SPLINE
SPL {X  -159.452, Y  +378.767, Z    +0.000, E1   +11.887, E3 +78162.676}
SPL {X  -159.840, Y  +384.856, Z    +0.000, E1    +7.126, E3 +78181.648}
SPL {X  -159.991, Y  +390.336, Z    +0.000, E1    +2.803, E3 +78195.471}
SPL {X  -160.000, Y  +403.532, Z    +0.000, E1    -6.523, E3 +78213.191}
SPL {X  -160.000, Y  +409.023, Z    +0.000, E1   -10.003, E3 +78223.965}
SPL {X  -160.000, Y  +418.032, Z    +0.000, E1   -14.569, E3 +78248.824}
SPL {X  -160.000, Y  +420.561, Z    +0.000, E1   -14.816, E3 +78266.304}
SPL {X  -160.000, Y  +422.801, Z    +0.000, E1   -14.823, E3 +78284.253}
SPL {X  -160.000, Y  +425.518, Z    +0.000, E1   -14.845, E3 +78306.027}
SPL {X  -160.000, Y  +428.688, Z    +0.000, E1   -14.854, E3 +78331.435}
SPL {X  -160.000, Y  +431.971, Z    +0.000, E1   -14.849, E3 +78357.904}
SPL {X  -160.000, Y  +435.345, Z    +0.000, E1   -14.857, E3 +78384.954}
SPL {X  -160.000, Y  +438.732, Z    +0.000, E1   -14.858, E3 +78412.103}
SPL {X  -160.000, Y  +441.925, Z    +0.000, E1   -14.848, E3 +78437.773}
SPL {X  -160.000, Y  +444.299, Z    +0.000, E1   -14.809, E3 +78456.958}
SPL {X  -160.000, Y  +446.229, Z    +0.000, E1   -14.820, E3 +78472.377}
SPL {X  -160.000, Y  +448.987, Z    +0.000, E1   -14.868, E3 +78494.313}
SPL {X  -160.000, Y  +452.351, Z    +0.000, E1   -14.871, E3 +78521.289}
SPL {X  -160.000, Y  +455.709, Z    +0.000, E1   -14.880, E3 +78548.103}
SPL {X  -160.000, Y  +458.189, Z    +0.000, E1   -14.832, E3 +78568.105}
SPL {X  -160.000, Y  +459.885, Z    +0.000, E1   -14.825, E3 +78581.776}
SPL {X  -160.000, Y  +462.438, Z    +0.000, E1   -14.868, E3 +78602.186}
SPL {X  -160.000, Y  +465.575, Z    +0.000, E1   -14.849, E3 +78627.494}
SPL {X  -160.000, Y  +468.581, Z    +0.000, E1   -14.841, E3 +78651.726}
SPL {X  -160.000, Y  +471.795, Z    +0.000, E1   -14.854, E3 +78677.514}
SPL {X  -160.000, Y  +475.138, Z    +0.000, E1   -14.853, E3 +78704.364}
SPL {X  -160.000, Y  +477.981, Z    +0.000, E1   -14.823, E3 +78727.284}
SPL {X  -160.000, Y  +480.658, Z    +0.000, E1   -14.835, E3 +78748.760}
SPL {X  -160.000, Y  +483.534, Z    +0.000, E1   -14.838, E3 +78771.855}
SPL {X  -160.000, Y  +486.226, Z    +0.000, E1   -14.823, E3 +78793.520}
SPL {X  -160.000, Y  +488.751, Z    +0.000, E1   -14.827, E3 +78813.793}
SPL {X  -160.000, Y  +491.612, Z    +0.000, E1   -14.844, E3 +78836.716}
SPL {X  -160.000, Y  +494.417, Z    +0.000, E1   -14.827, E3 +78859.306}
SPL {X  -160.000, Y  +496.961, Z    +0.000, E1   -14.824, E3 +78879.750}
SPL {X  -160.000, Y  +499.610, Z    +0.000, E1   -14.830, E3 +78901.023}
SPL {X  -160.000, Y  +502.268, Z    +0.000, E1   -14.832, E3 +78922.292}
SPL {X  -160.000, Y  +505.041, Z    +0.000, E1   -14.849, E3 +78944.455}
SPL {X  -160.000, Y  +507.743, Z    +0.000, E1   -14.842, E3 +78966.078}
SPL {X  -160.000, Y  +510.437, Z    +0.000, E1   -14.860, E3 +78987.592}
SPL {X  -160.000, Y  +513.179, Z    +0.000, E1   -14.849, E3 +79009.640}
SPL {X  -160.000, Y  +515.613, Z    +0.000, E1   -14.829, E3 +79029.310}
SPL {X  -160.000, Y  +518.188, Z    +0.000, E1   -14.845, E3 +79049.939}
SPL {X  -160.000, Y  +520.790, Z    +0.000, E1   -14.839, E3 +79070.768}
SPL {X  -160.000, Y  +523.469, Z    +0.000, E1   -14.855, E3 +79092.216}
SPL {X  -160.000, Y  +526.403, Z    +0.000, E1   -14.858, E3 +79115.753}
SPL {X  -160.000, Y  +529.266, Z    +0.000, E1   -14.848, E3 +79138.760}
SPL {X  -160.000, Y  +531.688, Z    +0.000, E1   -14.826, E3 +79158.310}
SPL {X  -160.000, Y  +534.214, Z    +0.000, E1   -14.841, E3 +79178.573}
SPL {X  -160.000, Y  +537.002, Z    +0.000, E1   -14.839, E3 +79200.991}
SPL {X  -160.000, Y  +539.729, Z    +0.000, E1   -14.840, E3 +79222.803}
SPL {X  -160.000, Y  +542.408, Z    +0.000, E1   -14.839, E3 +79244.356}
SPL {X  -160.000, Y  +545.014, Z    +0.000, E1   -14.831, E3 +79265.301}
SPL {X  -160.000, Y  +547.659, Z    +0.000, E1   -14.839, E3 +79286.515}
SPL {X  -160.000, Y  +550.215, Z    +0.000, E1   -14.827, E3 +79307.080}
SPL {X  -160.000, Y  +552.762, Z    +0.000, E1   -14.836, E3 +79327.499}
SPL {X  -160.000, Y  +555.331, Z    +0.000, E1   -14.837, E3 +79348.040}
SPL {X  -160.000, Y  +558.235, Z    +0.000, E1   -14.869, E3 +79371.203}
SPL {X  -160.000, Y  +561.088, Z    +0.000, E1   -14.848, E3 +79394.122}
SPL {X  -160.000, Y  +563.693, Z    +0.000, E1   -14.852, E3 +79414.982}
SPL {X  -160.000, Y  +566.560, Z    +0.000, E1   -14.865, E3 +79437.960}
SPL {X  -160.000, Y  +569.305, Z    +0.000, E1   -14.848, E3 +79459.988}
SPL {X  -160.000, Y  +571.769, Z    +0.000, E1   -14.852, E3 +79479.734}
SPL {X  -160.000, Y  +574.366, Z    +0.000, E1   -14.855, E3 +79500.521}
SPL {X  -160.000, Y  +577.037, Z    +0.000, E1   -14.859, E3 +79521.921}
SPL {X  -160.000, Y  +579.855, Z    +0.000, E1   -14.869, E3 +79544.448}
SPL {X  -160.000, Y  +582.456, Z    +0.000, E1   -14.854, E3 +79565.308}
SPL {X  -160.000, Y  +585.083, Z    +0.000, E1   -14.866, E3 +79586.358}
SPL {X  -160.000, Y  +587.675, Z    +0.000, E1   -14.853, E3 +79607.148}
SPL {X  -160.000, Y  +590.216, Z    +0.000, E1   -14.864, E3 +79627.468}
SPL {X  -160.000, Y  +592.848, Z    +0.000, E1   -14.865, E3 +79648.519}
SPL {X  -160.000, Y  +595.342, Z    +0.000, E1   -14.848, E3 +79668.696}
SPL {X  -160.000, Y  +597.995, Z    +0.000, E1   -14.848, E3 +79690.036}
SPL {X  -160.000, Y  +600.731, Z    +0.000, E1   -14.846, E3 +79711.988}
SPL {X  -160.000, Y  +603.404, Z    +0.000, E1   -14.846, E3 +79733.424}
SPL {X  -160.000, Y  +605.923, Z    +0.000, E1   -14.838, E3 +79753.664}
SPL {X  -160.000, Y  +608.492, Z    +0.000, E1   -14.846, E3 +79774.268}
SPL {X  -160.000, Y  +611.345, Z    +0.000, E1   -14.856, E3 +79797.126}
SPL {X  -160.000, Y  +614.087, Z    +0.000, E1   -14.839, E3 +79819.186}
SPL {X  -160.000, Y  +616.566, Z    +0.000, E1   -14.839, E3 +79839.079}
SPL {X  -160.000, Y  +619.350, Z    +0.000, E1   -14.855, E3 +79861.367}
SPL {X  -160.000, Y  +622.198, Z    +0.000, E1   -14.846, E3 +79884.252}
SPL {X  -160.000, Y  +624.642, Z    +0.000, E1   -14.829, E3 +79903.925}
SPL {X  -160.000, Y  +627.119, Z    +0.000, E1   -14.843, E3 +79923.764}
SPL {X  -160.000, Y  +629.682, Z    +0.000, E1   -14.838, E3 +79944.333}
SPL {X  -160.000, Y  +632.223, Z    +0.000, E1   -14.841, E3 +79964.725}
SPL {X  -160.000, Y  +634.941, Z    +0.000, E1   -14.846, E3 +79986.522}
SPL {X  -160.000, Y  +637.723, Z    +0.000, E1   -14.844, E3 +80008.867}
SPL {X  -160.000, Y  +640.315, Z    +0.000, E1   -14.836, E3 +80029.664}
SPL {X  -160.000, Y  +643.085, Z    +0.000, E1   -14.865, E3 +80051.716}
SPL {X  -160.000, Y  +645.845, Z    +0.000, E1   -14.848, E3 +80073.904}
SPL {X  -160.000, Y  +648.229, Z    +0.000, E1   -14.834, E3 +80093.113}
SPL {X  -160.000, Y  +650.656, Z    +0.000, E1   -14.835, E3 +80112.670}
SPL {X  -160.000, Y  +653.134, Z    +0.000, E1   -14.827, E3 +80132.597}
SPL {X  -160.000, Y  +655.670, Z    +0.000, E1   -14.841, E3 +80152.891}
SPL {X  -160.000, Y  +658.349, Z    +0.000, E1   -14.842, E3 +80174.367}
SPL {X  -160.000, Y  +660.936, Z    +0.000, E1   -14.838, E3 +80195.118}
SPL {X  -160.000, Y  +663.567, Z    +0.000, E1   -14.845, E3 +80216.249}
SPL {X  -160.000, Y  +666.216, Z    +0.000, E1   -14.832, E3 +80237.565}
SPL {X  -159.997, Y  +668.731, Z    +0.000, E1   -14.834, E3 +80257.757}
SPL {X  -159.962, Y  +671.176, Z    +0.000, E1   -14.822, E3 +80277.469}
SPL {X  -159.895, Y  +673.507, Z    +0.000, E1   -14.821, E3 +80296.200}
SPL {X  -159.785, Y  +675.985, Z    +0.000, E1   -14.818, E3 +80316.201}
SPL {X  -159.627, Y  +678.622, Z    +0.000, E1   -14.804, E3 +80337.554}
SPL {X  -159.438, Y  +681.094, Z    +0.000, E1   -14.770, E3 +80357.726}
SPL {X  -159.262, Y  +683.054, Z    +0.000, E1   -14.719, E3 +80373.954}
ENDSPLINE

SPLINE
SPL {X  -159.661, Y  +678.114, Z    +0.000, E1    -9.575, E3 +80403.546}
SPL {X  -159.942, Y  +672.020, Z    +0.000, E1    -4.692, E3 +80422.173}
SPL {X  -160.000, Y  +664.971, Z    +0.000, E1    +0.516, E3 +80441.723}
SPL {X  -160.000, Y  +660.032, Z    +0.000, E1    +3.995, E3 +80453.666}
SPL {X  -160.000, Y  +652.280, Z    +0.000, E1    +8.913, E3 +80472.181}
SPL {X  -160.000, Y  +644.147, Z    +0.000, E1   +13.158, E3 +80495.731}
SPL {X  -160.000, Y  +641.594, Z    +0.000, E1   +13.488, E3 +80514.172}
SPL {X  -160.000, Y  +639.799, Z    +0.000, E1   +13.486, E3 +80530.082}
SPL {X  -160.000, Y  +637.896, Z    +0.000, E1   +13.493, E3 +80546.897}
SPL {X  -160.000, Y  +635.832, Z    +0.000, E1   +13.499, E3 +80565.156}
SPL {X  -160.000, Y  +633.839, Z    +0.000, E1   +13.489, E3 +80582.845}
SPL {X  -160.000, Y  +631.625, Z    +0.000, E1   +13.508, E3 +80602.386}
SPL {X  -160.000, Y  +629.417, Z    +0.000, E1   +13.491, E3 +80621.997}
SPL {X  -160.000, Y  +627.180, Z    +0.000, E1   +13.508, E3 +80641.751}
SPL {X  -160.000, Y  +624.970, Z    +0.000, E1   +13.490, E3 +80661.401}
SPL {X  -160.000, Y  +623.020, Z    +0.000, E1   +13.491, E3 +80678.631}
SPL {X  -160.000, Y  +620.888, Z    +0.000, E1   +13.501, E3 +80697.493}
SPL {X  -160.000, Y  +618.790, Z    +0.000, E1   +13.488, E3 +80716.116}
SPL {X  -160.000, Y  +616.631, Z    +0.000, E1   +13.504, E3 +80735.169}
SPL {X  -160.000, Y  +614.230, Z    +0.000, E1   +13.510, E3 +80756.365}
SPL {X  -160.000, Y  +612.132, Z    +0.000, E1   +13.485, E3 +80775.081}
SPL {X  -160.000, Y  +610.405, Z    +0.000, E1   +13.477, E3 +80790.455}
SPL {X  -160.000, Y  +608.437, Z    +0.000, E1   +13.502, E3 +80807.710}
SPL {X  -160.000, Y  +606.281, Z    +0.000, E1   +13.502, E3 +80826.728}
SPL {X  -160.000, Y  +604.124, Z    +0.000, E1   +13.513, E3 +80845.783}
SPL {X  -160.000, Y  +601.878, Z    +0.000, E1   +13.505, E3 +80865.680}
SPL {X  -160.000, Y  +599.648, Z    +0.000, E1   +13.506, E3 +80885.457}
SPL {X  -160.000, Y  +597.673, Z    +0.000, E1   +13.479, E3 +80903.131}
SPL {X  -160.000, Y  +595.601, Z    +0.000, E1   +13.499, E3 +80921.414}
SPL {X  -160.000, Y  +593.187, Z    +0.000, E1   +13.500, E3 +80942.794}
SPL {X  -160.000, Y  +591.079, Z    +0.000, E1   +13.483, E3 +80961.520}
SPL {X  -160.000, Y  +589.151, Z    +0.000, E1   +13.489, E3 +80978.571}
SPL {X  -160.000, Y  +586.908, Z    +0.000, E1   +13.501, E3 +80998.416}
SPL {X  -160.000, Y  +584.660, Z    +0.000, E1   +13.490, E3 +81018.358}
SPL {X  -160.000, Y  +582.409, Z    +0.000, E1   +13.499, E3 +81038.276}
SPL {X  -160.000, Y  +580.150, Z    +0.000, E1   +13.490, E3 +81058.323}
SPL {X  -160.000, Y  +577.953, Z    +0.000, E1   +13.493, E3 +81077.781}
SPL {X  -160.000, Y  +575.630, Z    +0.000, E1   +13.502, E3 +81098.265}
SPL {X  -160.000, Y  +573.418, Z    +0.000, E1   +13.502, E3 +81117.773}
SPL {X  -160.000, Y  +571.226, Z    +0.000, E1   +13.520, E3 +81136.982}
SPL {X  -160.000, Y  +569.166, Z    +0.000, E1   +13.512, E3 +81155.172}
SPL {X  -160.000, Y  +567.275, Z    +0.000, E1   +13.517, E3 +81171.840}
SPL {X  -160.000, Y  +565.259, Z    +0.000, E1   +13.523, E3 +81189.629}
SPL {X  -160.000, Y  +563.305, Z    +0.000, E1   +13.512, E3 +81206.967}
SPL {X  -160.000, Y  +561.240, Z    +0.000, E1   +13.521, E3 +81225.229}
SPL {X  -160.000, Y  +558.881, Z    +0.000, E1   +13.524, E3 +81246.071}
SPL {X  -160.000, Y  +556.697, Z    +0.000, E1   +13.510, E3 +81265.457}
SPL {X  -160.000, Y  +554.624, Z    +0.000, E1   +13.512, E3 +81283.788}
SPL {X  -160.000, Y  +552.465, Z    +0.000, E1   +13.514, E3 +81302.872}
SPL {X  -160.000, Y  +550.315, Z    +0.000, E1   +13.514, E3 +81321.866}
SPL {X  -160.000, Y  +548.056, Z    +0.000, E1   +13.519, E3 +81341.867}
SPL {X  -160.000, Y  +545.826, Z    +0.000, E1   +13.501, E3 +81361.744}
SPL {X  -160.000, Y  +543.677, Z    +0.000, E1   +13.502, E3 +81380.802}
SPL {X  -160.000, Y  +541.664, Z    +0.000, E1   +13.489, E3 +81398.688}
SPL {X  -160.000, Y  +539.659, Z    +0.000, E1   +13.494, E3 +81416.448}
SPL {X  -160.000, Y  +537.370, Z    +0.000, E1   +13.501, E3 +81436.687}
SPL {X  -160.000, Y  +535.056, Z    +0.000, E1   +13.506, E3 +81457.082}
SPL {X  -160.000, Y  +532.975, Z    +0.000, E1   +13.494, E3 +81475.569}
SPL {X  -160.000, Y  +530.925, Z    +0.000, E1   +13.499, E3 +81493.731}
SPL {X  -160.000, Y  +528.768, Z    +0.000, E1   +13.498, E3 +81512.832}
SPL {X  -160.000, Y  +526.547, Z    +0.000, E1   +13.499, E3 +81532.501}
SPL {X  -160.000, Y  +523.964, Z    +0.000, E1   +13.742, E3 +81552.005}
SPL {X  -160.000, Y  +513.971, Z    +0.000, E1   +18.644, E3 +81570.917}
SPL {X  -160.000, Y  +513.562, Z    +0.000, E1   +16.972, E3 +81590.794}
SPL {X  -160.000, Y  +513.358, Z    +0.000, E1   +15.267, E3 +81611.066}
SPL {X  -160.000, Y  +512.244, Z    +0.000, E1   +14.473, E3 +81629.522}
SPL {X  -160.000, Y  +509.675, Z    +0.000, E1   +14.481, E3 +81650.666}
SPL {X  -160.000, Y  +507.162, Z    +0.000, E1   +14.470, E3 +81671.406}
SPL {X  -160.000, Y  +504.735, Z    +0.000, E1   +14.473, E3 +81691.377}
SPL {X  -160.000, Y  +502.261, Z    +0.000, E1   +14.476, E3 +81711.713}
SPL {X  -160.000, Y  +499.798, Z    +0.000, E1   +14.482, E3 +81731.916}
SPL {X  -160.000, Y  +497.435, Z    +0.000, E1   +14.476, E3 +81751.392}
SPL {X  -160.000, Y  +495.089, Z    +0.000, E1   +14.475, E3 +81770.759}
SPL {X  -160.000, Y  +492.764, Z    +0.000, E1   +14.469, E3 +81789.931}
SPL {X  -160.000, Y  +490.292, Z    +0.000, E1   +14.476, E3 +81810.332}
SPL {X  -160.000, Y  +487.641, Z    +0.000, E1   +14.470, E3 +81832.228}
SPL {X  -160.000, Y  +485.054, Z    +0.000, E1   +14.460, E3 +81853.670}
SPL {X  -160.000, Y  +482.421, Z    +0.000, E1   +14.461, E3 +81875.389}
SPL {X  -160.000, Y  +480.000, Z    +0.000, E1   +14.451, E3 +81895.353}
SPL {X  -160.000, Y  +477.551, Z    +0.000, E1   +14.466, E3 +81915.481}
SPL {X  -160.000, Y  +475.253, Z    +0.000, E1   +14.450, E3 +81934.455}
SPL {X  -160.000, Y  +473.070, Z    +0.000, E1   +14.454, E3 +81952.476}
SPL {X  -160.000, Y  +470.603, Z    +0.000, E1   +14.464, E3 +81972.777}
SPL {X  -160.000, Y  +468.243, Z    +0.000, E1   +14.458, E3 +81992.176}
SPL {X  -160.000, Y  +465.791, Z    +0.000, E1   +14.475, E3 +82012.320}
SPL {X  -160.000, Y  +463.103, Z    +0.000, E1   +14.474, E3 +82034.469}
SPL {X  -160.000, Y  +460.743, Z    +0.000, E1   +14.465, E3 +82053.877}
SPL {X  -160.000, Y  +458.292, Z    +0.000, E1   +14.492, E3 +82073.876}
SPL {X  -160.000, Y  +455.874, Z    +0.000, E1   +14.484, E3 +82093.734}
SPL {X  -160.000, Y  +453.555, Z    +0.000, E1   +14.488, E3 +82112.813}
SPL {X  -160.000, Y  +451.093, Z    +0.000, E1   +14.485, E3 +82133.125}
SPL {X  -160.000, Y  +448.700, Z    +0.000, E1   +14.483, E3 +82152.815}
SPL {X  -160.000, Y  +446.277, Z    +0.000, E1   +14.485, E3 +82172.738}
SPL {X  -160.000, Y  +443.879, Z    +0.000, E1   +14.485, E3 +82192.476}
SPL {X  -160.000, Y  +441.447, Z    +0.000, E1   +14.485, E3 +82212.484}
SPL {X  -160.000, Y  +439.006, Z    +0.000, E1   +14.488, E3 +82232.567}
SPL {X  -160.000, Y  +436.311, Z    +0.000, E1   +14.498, E3 +82254.726}
SPL {X  -160.000, Y  +433.559, Z    +0.000, E1   +14.491, E3 +82277.395}
SPL {X  -160.000, Y  +431.162, Z    +0.000, E1   +14.479, E3 +82297.146}
SPL {X  -160.000, Y  +429.152, Z    +0.000, E1   +14.469, E3 +82313.728}
SPL {X  -160.000, Y  +426.863, Z    +0.000, E1   +14.490, E3 +82332.507}
SPL {X  -160.000, Y  +424.653, Z    +0.000, E1   +14.467, E3 +82350.766}
SPL {X  -160.000, Y  +422.337, Z    +0.000, E1   +14.492, E3 +82369.750}
SPL {X  -160.000, Y  +419.639, Z    +0.000, E1   +14.504, E3 +82391.790}
SPL {X  -160.000, Y  +417.127, Z    +0.000, E1   +14.501, E3 +82412.381}
SPL {X  -160.000, Y  +414.849, Z    +0.000, E1   +14.496, E3 +82431.115}
SPL {X  -160.000, Y  +412.396, Z    +0.000, E1   +14.505, E3 +82451.304}
SPL {X  -160.000, Y  +409.815, Z    +0.000, E1   +14.498, E3 +82472.559}
SPL {X  -160.000, Y  +407.614, Z    +0.000, E1   +14.484, E3 +82490.684}
SPL {X  -160.000, Y  +405.406, Z    +0.000, E1   +14.501, E3 +82508.747}
SPL {X  -160.000, Y  +402.958, Z    +0.000, E1   +14.500, E3 +82528.917}
SPL {X  -160.000, Y  +400.690, Z    +0.000, E1   +14.484, E3 +82547.629}
SPL {X  -160.000, Y  +398.391, Z    +0.000, E1   +14.502, E3 +82566.455}
SPL {X  -160.000, Y  +395.999, Z    +0.000, E1   +14.484, E3 +82586.245}
SPL {X  -160.000, Y  +393.685, Z    +0.000, E1   +14.486, E3 +82605.317}
SPL {X  -159.999, Y  +391.313, Z    +0.000, E1   +14.479, E3 +82624.899}
SPL {X  -159.970, Y  +388.900, Z    +0.000, E1   +14.480, E3 +82644.783}
SPL {X  -159.903, Y  +386.417, Z    +0.000, E1   +14.475, E3 +82665.288}
SPL {X  -159.796, Y  +383.921, Z    +0.000, E1   +14.466, E3 +82685.944}
SPL {X  -159.651, Y  +381.443, Z    +0.000, E1   +14.453, E3 +82706.491}
SPL {X  -159.474, Y  +379.042, Z    +0.000, E1   +14.434, E3 +82726.455}
SPL {X  -159.316, Y  +377.219, Z    +0.000, E1   +14.400, E3 +82741.684}
ENDSPLINE

SPLINE
SPL {X  -159.452, Y  +378.767, Z    +0.000, E1   +11.887, E3 +82762.673}
SPL {X  -159.840, Y  +384.856, Z    +0.000, E1    +7.126, E3 +82781.645}
SPL {X  -159.991, Y  +390.336, Z    +0.000, E1    +2.803, E3 +82795.467}
SPL {X  -160.000, Y  +403.532, Z    +0.000, E1    -6.523, E3 +82813.188}
SPL {X  -160.000, Y  +409.023, Z    +0.000, E1   -10.003, E3 +82823.962}
SPL {X  -160.000, Y  +418.032, Z    +0.000, E1   -14.569, E3 +82848.821}
SPL {X  -160.000, Y  +420.561, Z    +0.000, E1   -14.816, E3 +82866.301}
SPL {X  -160.000, Y  +422.801, Z    +0.000, E1   -14.823, E3 +82884.249}
SPL {X  -160.000, Y  +425.518, Z    +0.000, E1   -14.845, E3 +82906.024}
SPL {X  -160.000, Y  +428.688, Z    +0.000, E1   -14.854, E3 +82931.432}
SPL {X  -160.000, Y  +431.971, Z    +0.000, E1   -14.849, E3 +82957.901}
SPL {X  -160.000, Y  +435.345, Z    +0.000, E1   -14.857, E3 +82984.951}
SPL {X  -160.000, Y  +438.732, Z    +0.000, E1   -14.858, E3 +83012.099}
SPL {X  -160.000, Y  +441.925, Z    +0.000, E1   -14.848, E3 +83037.770}
SPL {X  -160.000, Y  +444.299, Z    +0.000, E1   -14.809, E3 +83056.954}
SPL {X  -160.000, Y  +446.229, Z    +0.000, E1   -14.820, E3 +83072.373}
SPL {X  -160.000, Y  +448.987, Z    +0.000, E1   -14.868, E3 +83094.310}
SPL {X  -160.000, Y  +452.351, Z    +0.000, E1   -14.871, E3 +83121.286}
SPL {X  -160.000, Y  +455.709, Z    +0.000, E1   -14.880, E3 +83148.100}
SPL {X  -160.000, Y  +458.189, Z    +0.000, E1   -14.832, E3 +83168.102}
SPL {X  -160.000, Y  +459.885, Z    +0.000, E1   -14.825, E3 +83181.773}
SPL {X  -160.000, Y  +462.438, Z    +0.000, E1   -14.868, E3 +83202.183}
SPL {X  -160.000, Y  +465.575, Z    +0.000, E1   -14.849, E3 +83227.491}
SPL {X  -160.000, Y  +468.581, Z    +0.000, E1   -14.841, E3 +83251.723}
SPL {X  -160.000, Y  +471.795, Z    +0.000, E1   -14.854, E3 +83277.511}
SPL {X  -160.000, Y  +475.138, Z    +0.000, E1   -14.853, E3 +83304.361}
SPL {X  -160.000, Y  +477.981, Z    +0.000, E1   -14.823, E3 +83327.281}
SPL {X  -160.000, Y  +480.658, Z    +0.000, E1   -14.835, E3 +83348.757}
SPL {X  -160.000, Y  +483.534, Z    +0.000, E1   -14.838, E3 +83371.852}
SPL {X  -160.000, Y  +486.226, Z    +0.000, E1   -14.823, E3 +83393.517}
SPL {X  -160.000, Y  +488.751, Z    +0.000, E1   -14.827, E3 +83413.790}
SPL {X  -160.000, Y  +491.612, Z    +0.000, E1   -14.844, E3 +83436.712}
SPL {X  -160.000, Y  +494.417, Z    +0.000, E1   -14.827, E3 +83459.303}
SPL {X  -160.000, Y  +496.961, Z    +0.000, E1   -14.824, E3 +83479.747}
SPL {X  -160.000, Y  +499.610, Z    +0.000, E1   -14.830, E3 +83501.020}
SPL {X  -160.000, Y  +502.268, Z    +0.000, E1   -14.832, E3 +83522.289}
SPL {X  -160.000, Y  +505.041, Z    +0.000, E1   -14.849, E3 +83544.451}
SPL {X  -160.000, Y  +507.743, Z    +0.000, E1   -14.842, E3 +83566.075}
SPL {X  -160.000, Y  +510.437, Z    +0.000, E1   -14.860, E3 +83587.589}
SPL {X  -160.000, Y  +513.179, Z    +0.000, E1   -14.849, E3 +83609.636}
SPL {X  -160.000, Y  +515.613, Z    +0.000, E1   -14.829, E3 +83629.307}
SPL {X  -160.000, Y  +518.188, Z    +0.000, E1   -14.845, E3 +83649.936}
SPL {X  -160.000, Y  +520.790, Z    +0.000, E1   -14.839, E3 +83670.765}
SPL {X  -160.000, Y  +523.469, Z    +0.000, E1   -14.855, E3 +83692.213}
SPL {X  -160.000, Y  +526.403, Z    +0.000, E1   -14.858, E3 +83715.750}
SPL {X  -160.000, Y  +529.266, Z    +0.000, E1   -14.848, E3 +83738.757}
SPL {X  -160.000, Y  +531.688, Z    +0.000, E1   -14.826, E3 +83758.307}
SPL {X  -160.000, Y  +534.214, Z    +0.000, E1   -14.841, E3 +83778.570}
SPL {X  -160.000, Y  +537.002, Z    +0.000, E1   -14.839, E3 +83800.988}
SPL {X  -160.000, Y  +539.729, Z    +0.000, E1   -14.840, E3 +83822.799}
SPL {X  -160.000, Y  +542.408, Z    +0.000, E1   -14.839, E3 +83844.352}
SPL {X  -160.000, Y  +545.014, Z    +0.000, E1   -14.831, E3 +83865.298}
SPL {X  -160.000, Y  +547.659, Z    +0.000, E1   -14.839, E3 +83886.512}
SPL {X  -160.000, Y  +550.215, Z    +0.000, E1   -14.827, E3 +83907.077}
SPL {X  -160.000, Y  +552.762, Z    +0.000, E1   -14.836, E3 +83927.495}
SPL {X  -160.000, Y  +555.331, Z    +0.000, E1   -14.837, E3 +83948.036}
SPL {X  -160.000, Y  +558.235, Z    +0.000, E1   -14.869, E3 +83971.200}
SPL {X  -160.000, Y  +561.088, Z    +0.000, E1   -14.848, E3 +83994.119}
SPL {X  -160.000, Y  +563.693, Z    +0.000, E1   -14.852, E3 +84014.979}
SPL {X  -160.000, Y  +566.560, Z    +0.000, E1   -14.865, E3 +84037.957}
SPL {X  -160.000, Y  +569.305, Z    +0.000, E1   -14.848, E3 +84059.985}
SPL {X  -160.000, Y  +571.769, Z    +0.000, E1   -14.852, E3 +84079.731}
SPL {X  -160.000, Y  +574.366, Z    +0.000, E1   -14.855, E3 +84100.518}
SPL {X  -160.000, Y  +577.037, Z    +0.000, E1   -14.859, E3 +84121.917}
SPL {X  -160.000, Y  +579.855, Z    +0.000, E1   -14.869, E3 +84144.445}
SPL {X  -160.000, Y  +582.456, Z    +0.000, E1   -14.854, E3 +84165.305}
SPL {X  -160.000, Y  +585.083, Z    +0.000, E1   -14.866, E3 +84186.354}
SPL {X  -160.000, Y  +587.675, Z    +0.000, E1   -14.853, E3 +84207.145}
SPL {X  -160.000, Y  +590.216, Z    +0.000, E1   -14.864, E3 +84227.464}
SPL {X  -160.000, Y  +592.848, Z    +0.000, E1   -14.865, E3 +84248.516}
SPL {X  -160.000, Y  +595.342, Z    +0.000, E1   -14.848, E3 +84268.693}
SPL {X  -160.000, Y  +597.995, Z    +0.000, E1   -14.848, E3 +84290.033}
SPL {X  -160.000, Y  +600.731, Z    +0.000, E1   -14.846, E3 +84311.985}
SPL {X  -160.000, Y  +603.404, Z    +0.000, E1   -14.846, E3 +84333.420}
SPL {X  -160.000, Y  +605.923, Z    +0.000, E1   -14.838, E3 +84353.661}
SPL {X  -160.000, Y  +608.492, Z    +0.000, E1   -14.846, E3 +84374.265}
SPL {X  -160.000, Y  +611.345, Z    +0.000, E1   -14.856, E3 +84397.123}
SPL {X  -160.000, Y  +614.087, Z    +0.000, E1   -14.839, E3 +84419.182}
SPL {X  -160.000, Y  +616.566, Z    +0.000, E1   -14.839, E3 +84439.076}
SPL {X  -160.000, Y  +619.350, Z    +0.000, E1   -14.855, E3 +84461.364}
SPL {X  -160.000, Y  +622.198, Z    +0.000, E1   -14.846, E3 +84484.249}
SPL {X  -160.000, Y  +624.642, Z    +0.000, E1   -14.829, E3 +84503.921}
SPL {X  -160.000, Y  +627.119, Z    +0.000, E1   -14.843, E3 +84523.761}
SPL {X  -160.000, Y  +629.682, Z    +0.000, E1   -14.838, E3 +84544.330}
SPL {X  -160.000, Y  +632.223, Z    +0.000, E1   -14.841, E3 +84564.721}
SPL {X  -160.000, Y  +634.941, Z    +0.000, E1   -14.846, E3 +84586.519}
SPL {X  -160.000, Y  +637.723, Z    +0.000, E1   -14.844, E3 +84608.863}
SPL {X  -160.000, Y  +640.315, Z    +0.000, E1   -14.836, E3 +84629.661}
SPL {X  -160.000, Y  +643.085, Z    +0.000, E1   -14.865, E3 +84651.712}
SPL {X  -160.000, Y  +645.845, Z    +0.000, E1   -14.848, E3 +84673.900}
SPL {X  -160.000, Y  +648.229, Z    +0.000, E1   -14.834, E3 +84693.110}
SPL {X  -160.000, Y  +650.656, Z    +0.000, E1   -14.835, E3 +84712.667}
SPL {X  -160.000, Y  +653.134, Z    +0.000, E1   -14.827, E3 +84732.594}
SPL {X  -160.000, Y  +655.670, Z    +0.000, E1   -14.841, E3 +84752.888}
SPL {X  -160.000, Y  +658.349, Z    +0.000, E1   -14.842, E3 +84774.363}
SPL {X  -160.000, Y  +660.936, Z    +0.000, E1   -14.838, E3 +84795.115}
SPL {X  -160.000, Y  +663.567, Z    +0.000, E1   -14.845, E3 +84816.246}
SPL {X  -160.000, Y  +666.216, Z    +0.000, E1   -14.832, E3 +84837.562}
SPL {X  -159.997, Y  +668.731, Z    +0.000, E1   -14.834, E3 +84857.754}
SPL {X  -159.962, Y  +671.176, Z    +0.000, E1   -14.822, E3 +84877.465}
SPL {X  -159.895, Y  +673.507, Z    +0.000, E1   -14.821, E3 +84896.197}
SPL {X  -159.785, Y  +675.985, Z    +0.000, E1   -14.818, E3 +84916.198}
SPL {X  -159.627, Y  +678.622, Z    +0.000, E1   -14.804, E3 +84937.551}
SPL {X  -159.438, Y  +681.094, Z    +0.000, E1   -14.770, E3 +84957.722}
SPL {X  -159.262, Y  +683.054, Z    +0.000, E1   -14.719, E3 +84973.951}
ENDSPLINE

SPLINE
SPL {X  -159.661, Y  +678.114, Z    +0.000, E1    -9.575, E3 +85003.543}
SPL {X  -159.942, Y  +672.020, Z    +0.000, E1    -4.692, E3 +85022.169}
SPL {X  -160.000, Y  +664.971, Z    +0.000, E1    +0.516, E3 +85041.720}
SPL {X  -160.000, Y  +660.032, Z    +0.000, E1    +3.995, E3 +85053.663}
SPL {X  -160.000, Y  +652.280, Z    +0.000, E1    +8.913, E3 +85072.178}
SPL {X  -160.000, Y  +644.147, Z    +0.000, E1   +13.158, E3 +85095.728}
SPL {X  -160.000, Y  +641.594, Z    +0.000, E1   +13.488, E3 +85114.169}
SPL {X  -160.000, Y  +639.799, Z    +0.000, E1   +13.486, E3 +85130.079}
SPL {X  -160.000, Y  +637.896, Z    +0.000, E1   +13.493, E3 +85146.894}
SPL {X  -160.000, Y  +635.832, Z    +0.000, E1   +13.499, E3 +85165.153}
SPL {X  -160.000, Y  +633.839, Z    +0.000, E1   +13.489, E3 +85182.842}
SPL {X  -160.000, Y  +631.625, Z    +0.000, E1   +13.508, E3 +85202.382}
SPL {X  -160.000, Y  +629.417, Z    +0.000, E1   +13.491, E3 +85221.994}
SPL {X  -160.000, Y  +627.180, Z    +0.000, E1   +13.508, E3 +85241.748}
SPL {X  -160.000, Y  +624.970, Z    +0.000, E1   +13.490, E3 +85261.398}
SPL {X  -160.000, Y  +623.020, Z    +0.000, E1   +13.491, E3 +85278.628}
SPL {X  -160.000, Y  +620.888, Z    +0.000, E1   +13.501, E3 +85297.490}
SPL {X  -160.000, Y  +618.790, Z    +0.000, E1   +13.488, E3 +85316.112}
SPL {X  -160.000, Y  +616.631, Z    +0.000, E1   +13.504, E3 +85335.166}
SPL {X  -160.000, Y  +614.230, Z    +0.000, E1   +13.510, E3 +85356.362}
SPL {X  -160.000, Y  +612.132, Z    +0.000, E1   +13.485, E3 +85375.078}
SPL {X  -160.000, Y  +610.405, Z    +0.000, E1   +13.477, E3 +85390.452}
SPL {X  -160.000, Y  +608.437, Z    +0.000, E1   +13.502, E3 +85407.707}
SPL {X  -160.000, Y  +606.281, Z    +0.000, E1   +13.502, E3 +85426.725}
SPL {X  -160.000, Y  +604.124, Z    +0.000, E1   +13.513, E3 +85445.780}
SPL {X  -160.000, Y  +601.878, Z    +0.000, E1   +13.505, E3 +85465.677}
SPL {X  -160.000, Y  +599.648, Z    +0.000, E1   +13.506, E3 +85485.454}
SPL {X  -160.000, Y  +597.673, Z    +0.000, E1   +13.479, E3 +85503.127}
SPL {X  -160.000, Y  +595.601, Z    +0.000, E1   +13.499, E3 +85521.411}
SPL {X  -160.000, Y  +593.187, Z    +0.000, E1   +13.500, E3 +85542.791}
SPL {X  -160.000, Y  +591.079, Z    +0.000, E1   +13.483, E3 +85561.517}
SPL {X  -160.000, Y  +589.151, Z    +0.000, E1   +13.489, E3 +85578.568}
SPL {X  -160.000, Y  +586.908, Z    +0.000, E1   +13.501, E3 +85598.413}
SPL {X  -160.000, Y  +584.660, Z    +0.000, E1   +13.490, E3 +85618.355}
SPL {X  -160.000, Y  +582.409, Z    +0.000, E1   +13.499, E3 +85638.273}
SPL {X  -160.000, Y  +580.150, Z    +0.000, E1   +13.490, E3 +85658.320}
SPL {X  -160.000, Y  +577.953, Z    +0.000, E1   +13.493, E3 +85677.778}
SPL {X  -160.000, Y  +575.630, Z    +0.000, E1   +13.502, E3 +85698.262}
SPL {X  -160.000, Y  +573.418, Z    +0.000, E1   +13.502, E3 +85717.770}
SPL {X  -160.000, Y  +571.226, Z    +0.000, E1   +13.520, E3 +85736.979}
SPL {X  -160.000, Y  +569.166, Z    +0.000, E1   +13.512, E3 +85755.169}
SPL {X  -160.000, Y  +567.275, Z    +0.000, E1   +13.517, E3 +85771.836}
SPL {X  -160.000, Y  +565.259, Z    +0.000, E1   +13.523, E3 +85789.625}
SPL {X  -160.000, Y  +563.305, Z    +0.000, E1   +13.512, E3 +85806.964}
SPL {X  -160.000, Y  +561.240, Z    +0.000, E1   +13.521, E3 +85825.225}
SPL {X  -160.000, Y  +558.881, Z    +0.000, E1   +13.524, E3 +85846.068}
SPL {X  -160.000, Y  +556.697, Z    +0.000, E1   +13.510, E3 +85865.454}
SPL {X  -160.000, Y  +554.624, Z    +0.000, E1   +13.512, E3 +85883.785}
SPL {X  -160.000, Y  +552.465, Z    +0.000, E1   +13.514, E3 +85902.869}
SPL {X  -160.000, Y  +550.315, Z    +0.000, E1   +13.514, E3 +85921.863}
SPL {X  -160.000, Y  +548.056, Z    +0.000, E1   +13.519, E3 +85941.863}
SPL {X  -160.000, Y  +545.826, Z    +0.000, E1   +13.501, E3 +85961.741}
SPL {X  -160.000, Y  +543.677, Z    +0.000, E1   +13.502, E3 +85980.799}
SPL {X  -160.000, Y  +541.664, Z    +0.000, E1   +13.489, E3 +85998.684}
SPL {X  -160.000, Y  +539.659, Z    +0.000, E1   +13.494, E3 +86016.445}
SPL {X  -160.000, Y  +537.370, Z    +0.000, E1   +13.501, E3 +86036.684}
SPL {X  -160.000, Y  +535.056, Z    +0.000, E1   +13.506, E3 +86057.079}
SPL {X  -160.000, Y  +532.975, Z    +0.000, E1   +13.494, E3 +86075.566}
SPL {X  -160.000, Y  +530.925, Z    +0.000, E1   +13.499, E3 +86093.728}
SPL {X  -160.000, Y  +528.768, Z    +0.000, E1   +13.498, E3 +86112.829}
SPL {X  -160.000, Y  +526.547, Z    +0.000, E1   +13.499, E3 +86132.498}
SPL {X  -160.000, Y  +523.964, Z    +0.000, E1   +13.742, E3 +86152.002}
SPL {X  -160.000, Y  +513.971, Z    +0.000, E1   +18.644, E3 +86170.914}
SPL {X  -160.000, Y  +513.562, Z    +0.000, E1   +16.972, E3 +86190.791}
SPL {X  -160.000, Y  +513.358, Z    +0.000, E1   +15.267, E3 +86211.063}
SPL {X  -160.000, Y  +512.244, Z    +0.000, E1   +14.473, E3 +86229.519}
SPL {X  -160.000, Y  +509.675, Z    +0.000, E1   +14.481, E3 +86250.663}
SPL {X  -160.000, Y  +507.162, Z    +0.000, E1   +14.470, E3 +86271.403}
SPL {X  -160.000, Y  +504.735, Z    +0.000, E1   +14.473, E3 +86291.374}
SPL {X  -160.000, Y  +502.261, Z    +0.000, E1   +14.476, E3 +86311.710}
SPL {X  -160.000, Y  +499.798, Z    +0.000, E1   +14.482, E3 +86331.912}
SPL {X  -160.000, Y  +497.435, Z    +0.000, E1   +14.476, E3 +86351.389}
SPL {X  -160.000, Y  +495.089, Z    +0.000, E1   +14.475, E3 +86370.756}
SPL {X  -160.000, Y  +492.764, Z    +0.000, E1   +14.469, E3 +86389.927}
SPL {X  -160.000, Y  +490.292, Z    +0.000, E1   +14.476, E3 +86410.328}
SPL {X  -160.000, Y  +487.641, Z    +0.000, E1   +14.470, E3 +86432.224}
SPL {X  -160.000, Y  +485.054, Z    +0.000, E1   +14.460, E3 +86453.667}
SPL {X  -160.000, Y  +482.421, Z    +0.000, E1   +14.461, E3 +86475.385}
SPL {X  -160.000, Y  +480.000, Z    +0.000, E1   +14.451, E3 +86495.350}
SPL {X  -160.000, Y  +477.551, Z    +0.000, E1   +14.466, E3 +86515.478}
SPL {X  -160.000, Y  +475.253, Z    +0.000, E1   +14.450, E3 +86534.452}
SPL {X  -160.000, Y  +473.070, Z    +0.000, E1   +14.454, E3 +86552.473}
SPL {X  -160.000, Y  +470.603, Z    +0.000, E1   +14.464, E3 +86572.773}
SPL {X  -160.000, Y  +468.243, Z    +0.000, E1   +14.458, E3 +86592.173}
SPL {X  -160.000, Y  +465.791, Z    +0.000, E1   +14.475, E3 +86612.317}
SPL {X  -160.000, Y  +463.103, Z    +0.000, E1   +14.474, E3 +86634.465}
SPL {X  -160.000, Y  +460.743, Z    +0.000, E1   +14.465, E3 +86653.874}
SPL {X  -160.000, Y  +458.292, Z    +0.000, E1   +14.492, E3 +86673.873}
SPL {X  -160.000, Y  +455.874, Z    +0.000, E1   +14.484, E3 +86693.731}
SPL {X  -160.000, Y  +453.555, Z    +0.000, E1   +14.488, E3 +86712.810}
SPL {X  -160.000, Y  +451.093, Z    +0.000, E1   +14.485, E3 +86733.122}
SPL {X  -160.000, Y  +448.700, Z    +0.000, E1   +14.483, E3 +86752.811}
SPL {X  -160.000, Y  +446.277, Z    +0.000, E1   +14.485, E3 +86772.735}
SPL {X  -160.000, Y  +443.879, Z    +0.000, E1   +14.485, E3 +86792.473}
SPL {X  -160.000, Y  +441.447, Z    +0.000, E1   +14.485, E3 +86812.480}
SPL {X  -160.000, Y  +439.006, Z    +0.000, E1   +14.488, E3 +86832.563}
SPL {X  -160.000, Y  +436.311, Z    +0.000, E1   +14.498, E3 +86854.722}
SPL {X  -160.000, Y  +433.559, Z    +0.000, E1   +14.491, E3 +86877.392}
SPL {X  -160.000, Y  +431.162, Z    +0.000, E1   +14.479, E3 +86897.143}
SPL {X  -160.000, Y  +429.152, Z    +0.000, E1   +14.469, E3 +86913.724}
SPL {X  -160.000, Y  +426.863, Z    +0.000, E1   +14.490, E3 +86932.503}
SPL {X  -160.000, Y  +424.653, Z    +0.000, E1   +14.467, E3 +86950.763}
SPL {X  -160.000, Y  +422.337, Z    +0.000, E1   +14.492, E3 +86969.747}
SPL {X  -160.000, Y  +419.639, Z    +0.000, E1   +14.504, E3 +86991.787}
SPL {X  -160.000, Y  +417.127, Z    +0.000, E1   +14.501, E3 +87012.378}
SPL {X  -160.000, Y  +414.849, Z    +0.000, E1   +14.496, E3 +87031.112}
SPL {X  -160.000, Y  +412.396, Z    +0.000, E1   +14.505, E3 +87051.301}
SPL {X  -160.000, Y  +409.815, Z    +0.000, E1   +14.498, E3 +87072.555}
SPL {X  -160.000, Y  +407.614, Z    +0.000, E1   +14.484, E3 +87090.681}
SPL {X  -160.000, Y  +405.406, Z    +0.000, E1   +14.501, E3 +87108.744}
SPL {X  -160.000, Y  +402.958, Z    +0.000, E1   +14.500, E3 +87128.914}
SPL {X  -160.000, Y  +400.690, Z    +0.000, E1   +14.484, E3 +87147.625}
SPL {X  -160.000, Y  +398.391, Z    +0.000, E1   +14.502, E3 +87166.451}
SPL {X  -160.000, Y  +395.999, Z    +0.000, E1   +14.484, E3 +87186.241}
SPL {X  -160.000, Y  +393.685, Z    +0.000, E1   +14.486, E3 +87205.314}
SPL {X  -159.999, Y  +391.313, Z    +0.000, E1   +14.479, E3 +87224.896}
SPL {X  -159.970, Y  +388.900, Z    +0.000, E1   +14.480, E3 +87244.780}
SPL {X  -159.903, Y  +386.417, Z    +0.000, E1   +14.475, E3 +87265.285}
SPL {X  -159.796, Y  +383.921, Z    +0.000, E1   +14.466, E3 +87285.941}
SPL {X  -159.651, Y  +381.443, Z    +0.000, E1   +14.453, E3 +87306.488}
SPL {X  -159.474, Y  +379.042, Z    +0.000, E1   +14.434, E3 +87326.452}
SPL {X  -159.316, Y  +377.219, Z    +0.000, E1   +14.400, E3 +87341.681}
ENDSPLINE

SPLINE
SPL {X  -159.452, Y  +378.767, Z    +0.000, E1   +11.887, E3 +87362.670}
SPL {X  -159.840, Y  +384.856, Z    +0.000, E1    +7.126, E3 +87381.641}
SPL {X  -159.991, Y  +390.336, Z    +0.000, E1    +2.803, E3 +87395.464}
SPL {X  -160.000, Y  +403.532, Z    +0.000, E1    -6.523, E3 +87413.185}
SPL {X  -160.000, Y  +409.023, Z    +0.000, E1   -10.003, E3 +87423.958}
SPL {X  -160.000, Y  +418.032, Z    +0.000, E1   -14.569, E3 +87448.818}
SPL {X  -160.000, Y  +420.561, Z    +0.000, E1   -14.816, E3 +87466.298}
SPL {X  -160.000, Y  +422.801, Z    +0.000, E1   -14.823, E3 +87484.246}
SPL {X  -160.000, Y  +425.518, Z    +0.000, E1   -14.845, E3 +87506.021}
SPL {X  -160.000, Y  +428.688, Z    +0.000, E1   -14.854, E3 +87531.429}
SPL {X  -160.000, Y  +431.971, Z    +0.000, E1   -14.849, E3 +87557.898}
SPL {X  -160.000, Y  +435.345, Z    +0.000, E1   -14.857, E3 +87584.948}
SPL {X  -160.000, Y  +438.732, Z    +0.000, E1   -14.858, E3 +87612.096}
SPL {X  -160.000, Y  +441.925, Z    +0.000, E1   -14.848, E3 +87637.767}
SPL {X  -160.000, Y  +444.299, Z    +0.000, E1   -14.809, E3 +87656.951}
SPL {X  -160.000, Y  +446.229, Z    +0.000, E1   -14.820, E3 +87672.370}
SPL {X  -160.000, Y  +448.987, Z    +0.000, E1   -14.868, E3 +87694.307}
SPL {X  -160.000, Y  +452.351, Z    +0.000, E1   -14.871, E3 +87721.283}
SPL {X  -160.000, Y  +455.709, Z    +0.000, E1   -14.880, E3 +87748.097}
SPL {X  -160.000, Y  +458.189, Z    +0.000, E1   -14.832, E3 +87768.099}
SPL {X  -160.000, Y  +459.885, Z    +0.000, E1   -14.825, E3 +87781.769}
SPL {X  -160.000, Y  +462.438, Z    +0.000, E1   -14.868, E3 +87802.179}
SPL {X  -160.000, Y  +465.575, Z    +0.000, E1   -14.849, E3 +87827.488}
SPL {X  -160.000, Y  +468.581, Z    +0.000, E1   -14.841, E3 +87851.720}
SPL {X  -160.000, Y  +471.795, Z    +0.000, E1   -14.854, E3 +87877.507}
SPL {X  -160.000, Y  +475.138, Z    +0.000, E1   -14.853, E3 +87904.358}
SPL {X  -160.000, Y  +477.981, Z    +0.000, E1   -14.823, E3 +87927.278}
SPL {X  -160.000, Y  +480.658, Z    +0.000, E1   -14.835, E3 +87948.754}
SPL {X  -160.000, Y  +483.534, Z    +0.000, E1   -14.838, E3 +87971.849}
SPL {X  -160.000, Y  +486.226, Z    +0.000, E1   -14.823, E3 +87993.514}
SPL {X  -160.000, Y  +488.751, Z    +0.000, E1   -14.827, E3 +88013.786}
SPL {X  -160.000, Y  +491.612, Z    +0.000, E1   -14.844, E3 +88036.709}
SPL {X  -160.000, Y  +494.417, Z    +0.000, E1   -14.827, E3 +88059.300}
SPL {X  -160.000, Y  +496.961, Z    +0.000, E1   -14.824, E3 +88079.744}
SPL {X  -160.000, Y  +499.610, Z    +0.000, E1   -14.830, E3 +88101.016}
SPL {X  -160.000, Y  +502.268, Z    +0.000, E1   -14.832, E3 +88122.286}
SPL {X  -160.000, Y  +505.041, Z    +0.000, E1   -14.849, E3 +88144.448}
SPL {X  -160.000, Y  +507.743, Z    +0.000, E1   -14.842, E3 +88166.072}
SPL {X  -160.000, Y  +510.437, Z    +0.000, E1   -14.860, E3 +88187.586}
SPL {X  -160.000, Y  +513.179, Z    +0.000, E1   -14.849, E3 +88209.633}
SPL {X  -160.000, Y  +515.613, Z    +0.000, E1   -14.829, E3 +88229.304}
SPL {X  -160.000, Y  +518.188, Z    +0.000, E1   -14.845, E3 +88249.933}
SPL {X  -160.000, Y  +520.790, Z    +0.000, E1   -14.839, E3 +88270.762}
SPL {X  -160.000, Y  +523.469, Z    +0.000, E1   -14.855, E3 +88292.210}
SPL {X  -160.000, Y  +526.403, Z    +0.000, E1   -14.858, E3 +88315.746}
SPL {X  -160.000, Y  +529.266, Z    +0.000, E1   -14.848, E3 +88338.754}
SPL {X  -160.000, Y  +531.688, Z    +0.000, E1   -14.826, E3 +88358.303}
SPL {X  -160.000, Y  +534.214, Z    +0.000, E1   -14.841, E3 +88378.566}
SPL {X  -160.000, Y  +537.002, Z    +0.000, E1   -14.839, E3 +88400.985}
SPL {X  -160.000, Y  +539.729, Z    +0.000, E1   -14.840, E3 +88422.796}
SPL {X  -160.000, Y  +542.408, Z    +0.000, E1   -14.839, E3 +88444.349}
SPL {X  -160.000, Y  +545.014, Z    +0.000, E1   -14.831, E3 +88465.294}
SPL {X  -160.000, Y  +547.659, Z    +0.000, E1   -14.839, E3 +88486.509}
SPL {X  -160.000, Y  +550.215, Z    +0.000, E1   -14.827, E3 +88507.074}
SPL {X  -160.000, Y  +552.762, Z    +0.000, E1   -14.836, E3 +88527.492}
SPL {X  -160.000, Y  +555.331, Z    +0.000, E1   -14.837, E3 +88548.033}
SPL {X  -160.000, Y  +558.235, Z    +0.000, E1   -14.869, E3 +88571.197}
SPL {X  -160.000, Y  +561.088, Z    +0.000, E1   -14.848, E3 +88594.115}
SPL {X  -160.000, Y  +563.693, Z    +0.000, E1   -14.852, E3 +88614.976}
SPL {X  -160.000, Y  +566.560, Z    +0.000, E1   -14.865, E3 +88637.953}
SPL {X  -160.000, Y  +569.305, Z    +0.000, E1   -14.848, E3 +88659.982}
SPL {X  -160.000, Y  +571.769, Z    +0.000, E1   -14.852, E3 +88679.728}
SPL {X  -160.000, Y  +574.366, Z    +0.000, E1   -14.855, E3 +88700.515}
SPL {X  -160.000, Y  +577.037, Z    +0.000, E1   -14.859, E3 +88721.914}
SPL {X  -160.000, Y  +579.855, Z    +0.000, E1   -14.869, E3 +88744.441}
SPL {X  -160.000, Y  +582.456, Z    +0.000, E1   -14.854, E3 +88765.301}
SPL {X  -160.000, Y  +585.083, Z    +0.000, E1   -14.866, E3 +88786.351}
SPL {X  -160.000, Y  +587.675, Z    +0.000, E1   -14.853, E3 +88807.142}
SPL {X  -160.000, Y  +590.216, Z    +0.000, E1   -14.864, E3 +88827.461}
SPL {X  -160.000, Y  +592.848, Z    +0.000, E1   -14.865, E3 +88848.512}
SPL {X  -160.000, Y  +595.342, Z    +0.000, E1   -14.848, E3 +88868.690}
SPL {X  -160.000, Y  +597.995, Z    +0.000, E1   -14.848, E3 +88890.030}
SPL {X  -160.000, Y  +600.731, Z    +0.000, E1   -14.846, E3 +88911.981}
SPL {X  -160.000, Y  +603.404, Z    +0.000, E1   -14.846, E3 +88933.417}
SPL {X  -160.000, Y  +605.923, Z    +0.000, E1   -14.838, E3 +88953.658}
SPL {X  -160.000, Y  +608.492, Z    +0.000, E1   -14.846, E3 +88974.262}
SPL {X  -160.000, Y  +611.345, Z    +0.000, E1   -14.856, E3 +88997.120}
SPL {X  -160.000, Y  +614.087, Z    +0.000, E1   -14.839, E3 +89019.179}
SPL {X  -160.000, Y  +616.566, Z    +0.000, E1   -14.839, E3 +89039.073}
SPL {X  -160.000, Y  +619.350, Z    +0.000, E1   -14.855, E3 +89061.361}
SPL {X  -160.000, Y  +622.198, Z    +0.000, E1   -14.846, E3 +89084.246}
SPL {X  -160.000, Y  +624.642, Z    +0.000, E1   -14.829, E3 +89103.918}
SPL {X  -160.000, Y  +627.119, Z    +0.000, E1   -14.843, E3 +89123.758}
SPL {X  -160.000, Y  +629.682, Z    +0.000, E1   -14.838, E3 +89144.327}
SPL {X  -160.000, Y  +632.223, Z    +0.000, E1   -14.841, E3 +89164.718}
SPL {X  -160.000, Y  +634.941, Z    +0.000, E1   -14.846, E3 +89186.516}
SPL {X  -160.000, Y  +637.723, Z    +0.000, E1   -14.844, E3 +89208.860}
SPL {X  -160.000, Y  +640.315, Z    +0.000, E1   -14.836, E3 +89229.658}
SPL {X  -160.000, Y  +643.085, Z    +0.000, E1   -14.865, E3 +89251.709}
SPL {X  -160.000, Y  +645.845, Z    +0.000, E1   -14.848, E3 +89273.897}
SPL {X  -160.000, Y  +648.229, Z    +0.000, E1   -14.834, E3 +89293.107}
SPL {X  -160.000, Y  +650.656, Z    +0.000, E1   -14.835, E3 +89312.663}
SPL {X  -160.000, Y  +653.134, Z    +0.000, E1   -14.827, E3 +89332.590}
SPL {X  -160.000, Y  +655.670, Z    +0.000, E1   -14.841, E3 +89352.885}
SPL {X  -160.000, Y  +658.349, Z    +0.000, E1   -14.842, E3 +89374.360}
SPL {X  -160.000, Y  +660.936, Z    +0.000, E1   -14.838, E3 +89395.112}
SPL {X  -160.000, Y  +663.567, Z    +0.000, E1   -14.845, E3 +89416.242}
SPL {X  -160.000, Y  +666.216, Z    +0.000, E1   -14.832, E3 +89437.559}
SPL {X  -159.997, Y  +668.731, Z    +0.000, E1   -14.834, E3 +89457.751}
SPL {X  -159.962, Y  +671.176, Z    +0.000, E1   -14.822, E3 +89477.462}
SPL {X  -159.895, Y  +673.507, Z    +0.000, E1   -14.821, E3 +89496.193}
SPL {X  -159.785, Y  +675.985, Z    +0.000, E1   -14.818, E3 +89516.195}
SPL {X  -159.627, Y  +678.622, Z    +0.000, E1   -14.804, E3 +89537.548}
SPL {X  -159.438, Y  +681.094, Z    +0.000, E1   -14.770, E3 +89557.719}
SPL {X  -159.262, Y  +683.054, Z    +0.000, E1   -14.719, E3 +89573.947}
ENDSPLINE

SPLINE
SPL {X  -159.661, Y  +678.114, Z    +0.000, E1    -9.575, E3 +89603.539}
SPL {X  -159.942, Y  +672.020, Z    +0.000, E1    -4.692, E3 +89622.166}
SPL {X  -160.000, Y  +664.971, Z    +0.000, E1    +0.516, E3 +89641.717}
SPL {X  -160.000, Y  +660.032, Z    +0.000, E1    +3.995, E3 +89653.659}
SPL {X  -160.000, Y  +652.280, Z    +0.000, E1    +8.913, E3 +89672.174}
SPL {X  -160.000, Y  +644.147, Z    +0.000, E1   +13.158, E3 +89695.725}
SPL {X  -160.000, Y  +641.594, Z    +0.000, E1   +13.488, E3 +89714.166}
SPL {X  -160.000, Y  +639.799, Z    +0.000, E1   +13.486, E3 +89730.076}
SPL {X  -160.000, Y  +637.896, Z    +0.000, E1   +13.493, E3 +89746.891}
SPL {X  -160.000, Y  +635.832, Z    +0.000, E1   +13.499, E3 +89765.150}
SPL {X  -160.000, Y  +633.839, Z    +0.000, E1   +13.489, E3 +89782.838}
SPL {X  -160.000, Y  +631.625, Z    +0.000, E1   +13.508, E3 +89802.379}
SPL {X  -160.000, Y  +629.417, Z    +0.000, E1   +13.491, E3 +89821.991}
SPL {X  -160.000, Y  +627.180, Z    +0.000, E1   +13.508, E3 +89841.745}
SPL {X  -160.000, Y  +624.970, Z    +0.000, E1   +13.490, E3 +89861.395}
SPL {X  -160.000, Y  +623.020, Z    +0.000, E1   +13.491, E3 +89878.624}
SPL {X  -160.000, Y  +620.888, Z    +0.000, E1   +13.501, E3 +89897.487}
SPL {X  -160.000, Y  +618.790, Z    +0.000, E1   +13.488, E3 +89916.109}
SPL {X  -160.000, Y  +616.631, Z    +0.000, E1   +13.504, E3 +89935.163}
SPL {X  -160.000, Y  +614.230, Z    +0.000, E1   +13.510, E3 +89956.359}
SPL {X  -160.000, Y  +612.132, Z    +0.000, E1   +13.485, E3 +89975.075}
SPL {X  -160.000, Y  +610.405, Z    +0.000, E1   +13.477, E3 +89990.448}
SPL {X  -160.000, Y  +608.437, Z    +0.000, E1   +13.502, E3 +90007.704}
SPL {X  -160.000, Y  +606.281, Z    +0.000, E1   +13.502, E3 +90026.721}
SPL {X  -160.000, Y  +604.124, Z    +0.000, E1   +13.513, E3 +90045.777}
SPL {X  -160.000, Y  +601.878, Z    +0.000, E1   +13.505, E3 +90065.674}
SPL {X  -160.000, Y  +599.648, Z    +0.000, E1   +13.506, E3 +90085.451}
SPL {X  -160.000, Y  +597.673, Z    +0.000, E1   +13.479, E3 +90103.124}
SPL {X  -160.000, Y  +595.601, Z    +0.000, E1   +13.499, E3 +90121.407}
SPL {X  -160.000, Y  +593.187, Z    +0.000, E1   +13.500, E3 +90142.787}
SPL {X  -160.000, Y  +591.079, Z    +0.000, E1   +13.483, E3 +90161.514}
SPL {X  -160.000, Y  +589.151, Z    +0.000, E1   +13.489, E3 +90178.565}
SPL {X  -160.000, Y  +586.908, Z    +0.000, E1   +13.501, E3 +90198.410}
SPL {X  -160.000, Y  +584.660, Z    +0.000, E1   +13.490, E3 +90218.352}
SPL {X  -160.000, Y  +582.409, Z    +0.000, E1   +13.499, E3 +90238.270}
SPL {X  -160.000, Y  +580.150, Z    +0.000, E1   +13.490, E3 +90258.316}
SPL {X  -160.000, Y  +577.953, Z    +0.000, E1   +13.493, E3 +90277.775}
SPL {X  -160.000, Y  +575.630, Z    +0.000, E1   +13.502, E3 +90298.259}
SPL {X  -160.000, Y  +573.418, Z    +0.000, E1   +13.502, E3 +90317.767}
SPL {X  -160.000, Y  +571.226, Z    +0.000, E1   +13.520, E3 +90336.975}
SPL {X  -160.000, Y  +569.166, Z    +0.000, E1   +13.512, E3 +90355.166}
SPL {X  -160.000, Y  +567.275, Z    +0.000, E1   +13.517, E3 +90371.833}
SPL {X  -160.000, Y  +565.259, Z    +0.000, E1   +13.523, E3 +90389.622}
SPL {X  -160.000, Y  +563.305, Z    +0.000, E1   +13.512, E3 +90406.961}
SPL {X  -160.000, Y  +561.240, Z    +0.000, E1   +13.521, E3 +90425.222}
SPL {X  -160.000, Y  +558.881, Z    +0.000, E1   +13.524, E3 +90446.065}
SPL {X  -160.000, Y  +556.697, Z    +0.000, E1   +13.510, E3 +90465.451}
SPL {X  -160.000, Y  +554.624, Z    +0.000, E1   +13.512, E3 +90483.781}
SPL {X  -160.000, Y  +552.465, Z    +0.000, E1   +13.514, E3 +90502.866}
SPL {X  -160.000, Y  +550.315, Z    +0.000, E1   +13.514, E3 +90521.859}
SPL {X  -160.000, Y  +548.056, Z    +0.000, E1   +13.519, E3 +90541.860}
SPL {X  -160.000, Y  +545.826, Z    +0.000, E1   +13.501, E3 +90561.738}
SPL {X  -160.000, Y  +543.677, Z    +0.000, E1   +13.502, E3 +90580.796}
SPL {X  -160.000, Y  +541.664, Z    +0.000, E1   +13.489, E3 +90598.681}
SPL {X  -160.000, Y  +539.659, Z    +0.000, E1   +13.494, E3 +90616.441}
SPL {X  -160.000, Y  +537.370, Z    +0.000, E1   +13.501, E3 +90636.680}
SPL {X  -160.000, Y  +535.056, Z    +0.000, E1   +13.506, E3 +90657.076}
SPL {X  -160.000, Y  +532.975, Z    +0.000, E1   +13.494, E3 +90675.563}
SPL {X  -160.000, Y  +530.925, Z    +0.000, E1   +13.499, E3 +90693.724}
SPL {X  -160.000, Y  +528.768, Z    +0.000, E1   +13.498, E3 +90712.826}
SPL {X  -160.000, Y  +526.547, Z    +0.000, E1   +13.499, E3 +90732.494}
SPL {X  -160.000, Y  +523.964, Z    +0.000, E1   +13.742, E3 +90751.999}
SPL {X  -160.000, Y  +513.971, Z    +0.000, E1   +18.644, E3 +90770.911}
SPL {X  -160.000, Y  +513.562, Z    +0.000, E1   +16.972, E3 +90790.788}
SPL {X  -160.000, Y  +513.358, Z    +0.000, E1   +15.267, E3 +90811.060}
SPL {X  -160.000, Y  +512.244, Z    +0.000, E1   +14.473, E3 +90829.516}
SPL {X  -160.000, Y  +509.675, Z    +0.000, E1   +14.481, E3 +90850.659}
SPL {X  -160.000, Y  +507.162, Z    +0.000, E1   +14.470, E3 +90871.400}
SPL {X  -160.000, Y  +504.735, Z    +0.000, E1   +14.473, E3 +90891.371}
SPL {X  -160.000, Y  +502.261, Z    +0.000, E1   +14.476, E3 +90911.707}
SPL {X  -160.000, Y  +499.798, Z    +0.000, E1   +14.482, E3 +90931.909}
SPL {X  -160.000, Y  +497.435, Z    +0.000, E1   +14.476, E3 +90951.386}
SPL {X  -160.000, Y  +495.089, Z    +0.000, E1   +14.475, E3 +90970.753}
SPL {X  -160.000, Y  +492.764, Z    +0.000, E1   +14.469, E3 +90989.924}
SPL {X  -160.000, Y  +490.292, Z    +0.000, E1   +14.476, E3 +91010.325}
SPL {X  -160.000, Y  +487.641, Z    +0.000, E1   +14.470, E3 +91032.221}
SPL {X  -160.000, Y  +485.054, Z    +0.000, E1   +14.460, E3 +91053.664}
SPL {X  -160.000, Y  +482.421, Z    +0.000, E1   +14.461, E3 +91075.382}
SPL {X  -160.000, Y  +480.000, Z    +0.000, E1   +14.451, E3 +91095.346}
SPL {X  -160.000, Y  +477.551, Z    +0.000, E1   +14.466, E3 +91115.475}
SPL {X  -160.000, Y  +475.253, Z    +0.000, E1   +14.450, E3 +91134.449}
SPL {X  -160.000, Y  +473.070, Z    +0.000, E1   +14.454, E3 +91152.470}
SPL {X  -160.000, Y  +470.603, Z    +0.000, E1   +14.464, E3 +91172.770}
SPL {X  -160.000, Y  +468.243, Z    +0.000, E1   +14.458, E3 +91192.169}
SPL {X  -160.000, Y  +465.791, Z    +0.000, E1   +14.475, E3 +91212.314}
SPL {X  -160.000, Y  +463.103, Z    +0.000, E1   +14.474, E3 +91234.462}
SPL {X  -160.000, Y  +460.743, Z    +0.000, E1   +14.465, E3 +91253.871}
SPL {X  -160.000, Y  +458.292, Z    +0.000, E1   +14.492, E3 +91273.870}
SPL {X  -160.000, Y  +455.874, Z    +0.000, E1   +14.484, E3 +91293.727}
SPL {X  -160.000, Y  +453.555, Z    +0.000, E1   +14.488, E3 +91312.807}
SPL {X  -160.000, Y  +451.093, Z    +0.000, E1   +14.485, E3 +91333.119}
SPL {X  -160.000, Y  +448.700, Z    +0.000, E1   +14.483, E3 +91352.808}
SPL {X  -160.000, Y  +446.277, Z    +0.000, E1   +14.485, E3 +91372.732}
SPL {X  -160.000, Y  +443.879, Z    +0.000, E1   +14.485, E3 +91392.470}
SPL {X  -160.000, Y  +441.447, Z    +0.000, E1   +14.485, E3 +91412.477}
SPL {X  -160.000, Y  +439.006, Z    +0.000, E1   +14.488, E3 +91432.560}
SPL {X  -160.000, Y  +436.311, Z    +0.000, E1   +14.498, E3 +91454.719}
SPL {X  -160.000, Y  +433.559, Z    +0.000, E1   +14.491, E3 +91477.389}
SPL {X  -160.000, Y  +431.162, Z    +0.000, E1   +14.479, E3 +91497.140}
SPL {X  -160.000, Y  +429.152, Z    +0.000, E1   +14.469, E3 +91513.721}
SPL {X  -160.000, Y  +426.863, Z    +0.000, E1   +14.490, E3 +91532.500}
SPL {X  -160.000, Y  +424.653, Z    +0.000, E1   +14.467, E3 +91550.760}
SPL {X  -160.000, Y  +422.337, Z    +0.000, E1   +14.492, E3 +91569.744}
SPL {X  -160.000, Y  +419.639, Z    +0.000, E1   +14.504, E3 +91591.784}
SPL {X  -160.000, Y  +417.127, Z    +0.000, E1   +14.501, E3 +91612.375}
SPL {X  -160.000, Y  +414.849, Z    +0.000, E1   +14.496, E3 +91631.109}
SPL {X  -160.000, Y  +412.396, Z    +0.000, E1   +14.505, E3 +91651.298}
SPL {X  -160.000, Y  +409.815, Z    +0.000, E1   +14.498, E3 +91672.552}
SPL {X  -160.000, Y  +407.614, Z    +0.000, E1   +14.484, E3 +91690.677}
SPL {X  -160.000, Y  +405.406, Z    +0.000, E1   +14.501, E3 +91708.740}
SPL {X  -160.000, Y  +402.958, Z    +0.000, E1   +14.500, E3 +91728.911}
SPL {X  -160.000, Y  +400.690, Z    +0.000, E1   +14.484, E3 +91747.622}
SPL {X  -160.000, Y  +398.391, Z    +0.000, E1   +14.502, E3 +91766.448}
SPL {X  -160.000, Y  +395.999, Z    +0.000, E1   +14.484, E3 +91786.238}
SPL {X  -160.000, Y  +393.685, Z    +0.000, E1   +14.486, E3 +91805.310}
SPL {X  -159.999, Y  +391.313, Z    +0.000, E1   +14.479, E3 +91824.892}
SPL {X  -159.970, Y  +388.900, Z    +0.000, E1   +14.480, E3 +91844.777}
SPL {X  -159.903, Y  +386.417, Z    +0.000, E1   +14.475, E3 +91865.282}
SPL {X  -159.796, Y  +383.921, Z    +0.000, E1   +14.466, E3 +91885.937}
SPL {X  -159.651, Y  +381.443, Z    +0.000, E1   +14.453, E3 +91906.485}
SPL {X  -159.474, Y  +379.042, Z    +0.000, E1   +14.434, E3 +91926.449}
SPL {X  -159.316, Y  +377.219, Z    +0.000, E1   +14.400, E3 +91941.677}
ENDSPLINE

SPLINE
SPL {X  -159.452, Y  +378.767, Z    +0.000, E1   +11.887, E3 +91962.667}
SPL {X  -159.840, Y  +384.856, Z    +0.000, E1    +7.126, E3 +91981.638}
SPL {X  -159.991, Y  +390.336, Z    +0.000, E1    +2.803, E3 +91995.461}
SPL {X  -160.000, Y  +403.532, Z    +0.000, E1    -6.523, E3 +92013.182}
SPL {X  -160.000, Y  +409.023, Z    +0.000, E1   -10.003, E3 +92023.955}
SPL {X  -160.000, Y  +418.032, Z    +0.000, E1   -14.569, E3 +92048.814}
SPL {X  -160.000, Y  +420.561, Z    +0.000, E1   -14.816, E3 +92066.295}
SPL {X  -160.000, Y  +422.801, Z    +0.000, E1   -14.823, E3 +92084.243}
SPL {X  -160.000, Y  +425.518, Z    +0.000, E1   -14.845, E3 +92106.018}
SPL {X  -160.000, Y  +428.688, Z    +0.000, E1   -14.854, E3 +92131.426}
SPL {X  -160.000, Y  +431.971, Z    +0.000, E1   -14.849, E3 +92157.894}
SPL {X  -160.000, Y  +435.345, Z    +0.000, E1   -14.857, E3 +92184.945}
SPL {X  -160.000, Y  +438.732, Z    +0.000, E1   -14.858, E3 +92212.093}
SPL {X  -160.000, Y  +441.925, Z    +0.000, E1   -14.848, E3 +92237.763}
SPL {X  -160.000, Y  +444.299, Z    +0.000, E1   -14.809, E3 +92256.948}
SPL {X  -160.000, Y  +446.229, Z    +0.000, E1   -14.820, E3 +92272.367}
SPL {X  -160.000, Y  +448.987, Z    +0.000, E1   -14.868, E3 +92294.304}
SPL {X  -160.000, Y  +452.351, Z    +0.000, E1   -14.871, E3 +92321.280}
SPL {X  -160.000, Y  +455.709, Z    +0.000, E1   -14.880, E3 +92348.094}
SPL {X  -160.000, Y  +458.189, Z    +0.000, E1   -14.832, E3 +92368.095}
SPL {X  -160.000, Y  +459.885, Z    +0.000, E1   -14.825, E3 +92381.766}
SPL {X  -160.000, Y  +462.438, Z    +0.000, E1   -14.868, E3 +92402.176}
SPL {X  -160.000, Y  +465.575, Z    +0.000, E1   -14.849, E3 +92427.484}
SPL {X  -160.000, Y  +468.581, Z    +0.000, E1   -14.841, E3 +92451.717}
SPL {X  -160.000, Y  +471.795, Z    +0.000, E1   -14.854, E3 +92477.504}
SPL {X  -160.000, Y  +475.138, Z    +0.000, E1   -14.853, E3 +92504.355}
SPL {X  -160.000, Y  +477.981, Z    +0.000, E1   -14.823, E3 +92527.275}
SPL {X  -160.000, Y  +480.658, Z    +0.000, E1   -14.835, E3 +92548.751}
SPL {X  -160.000, Y  +483.534, Z    +0.000, E1   -14.838, E3 +92571.846}
SPL {X  -160.000, Y  +486.226, Z    +0.000, E1   -14.823, E3 +92593.511}
SPL {X  -160.000, Y  +488.751, Z    +0.000, E1   -14.827, E3 +92613.783}
SPL {X  -160.000, Y  +491.612, Z    +0.000, E1   -14.844, E3 +92636.706}
SPL {X  -160.000, Y  +494.417, Z    +0.000, E1   -14.827, E3 +92659.297}
SPL {X  -160.000, Y  +496.961, Z    +0.000, E1   -14.824, E3 +92679.741}
SPL {X  -160.000, Y  +499.610, Z    +0.000, E1   -14.830, E3 +92701.013}
SPL {X  -160.000, Y  +502.268, Z    +0.000, E1   -14.832, E3 +92722.282}
SPL {X  -160.000, Y  +505.041, Z    +0.000, E1   -14.849, E3 +92744.445}
SPL {X  -160.000, Y  +507.743, Z    +0.000, E1   -14.842, E3 +92766.069}
SPL {X  -160.000, Y  +510.437, Z    +0.000, E1   -14.860, E3 +92787.583}
SPL {X  -160.000, Y  +513.179, Z    +0.000, E1   -14.849, E3 +92809.630}
SPL {X  -160.000, Y  +515.613, Z    +0.000, E1   -14.829, E3 +92829.300}
SPL {X  -160.000, Y  +518.188, Z    +0.000, E1   -14.845, E3 +92849.930}
SPL {X  -160.000, Y  +520.790, Z    +0.000, E1   -14.839, E3 +92870.759}
SPL {X  -160.000, Y  +523.469, Z    +0.000, E1   -14.855, E3 +92892.207}
SPL {X  -160.000, Y  +526.403, Z    +0.000, E1   -14.858, E3 +92915.743}
SPL {X  -160.000, Y  +529.266, Z    +0.000, E1   -14.848, E3 +92938.751}
SPL {X  -160.000, Y  +531.688, Z    +0.000, E1   -14.826, E3 +92958.300}
SPL {X  -160.000, Y  +534.214, Z    +0.000, E1   -14.841, E3 +92978.563}
SPL {X  -160.000, Y  +537.002, Z    +0.000, E1   -14.839, E3 +93000.981}
SPL {X  -160.000, Y  +539.729, Z    +0.000, E1   -14.840, E3 +93022.793}
SPL {X  -160.000, Y  +542.408, Z    +0.000, E1   -14.839, E3 +93044.346}
SPL {X  -160.000, Y  +545.014, Z    +0.000, E1   -14.831, E3 +93065.291}
SPL {X  -160.000, Y  +547.659, Z    +0.000, E1   -14.839, E3 +93086.506}
SPL {X  -160.000, Y  +550.215, Z    +0.000, E1   -14.827, E3 +93107.071}
SPL {X  -160.000, Y  +552.762, Z    +0.000, E1   -14.836, E3 +93127.489}
SPL {X  -160.000, Y  +555.331, Z    +0.000, E1   -14.837, E3 +93148.030}
SPL {X  -160.000, Y  +558.235, Z    +0.000, E1   -14.869, E3 +93171.194}
SPL {X  -160.000, Y  +561.088, Z    +0.000, E1   -14.848, E3 +93194.112}
SPL {X  -160.000, Y  +563.693, Z    +0.000, E1   -14.852, E3 +93214.973}
SPL {X  -160.000, Y  +566.560, Z    +0.000, E1   -14.865, E3 +93237.950}
SPL {X  -160.000, Y  +569.305, Z    +0.000, E1   -14.848, E3 +93259.979}
SPL {X  -160.000, Y  +571.769, Z    +0.000, E1   -14.852, E3 +93279.724}
SPL {X  -160.000, Y  +574.366, Z    +0.000, E1   -14.855, E3 +93300.511}
SPL {X  -160.000, Y  +577.037, Z    +0.000, E1   -14.859, E3 +93321.911}
SPL {X  -160.000, Y  +579.855, Z    +0.000, E1   -14.869, E3 +93344.438}
SPL {X  -160.000, Y  +582.456, Z    +0.000, E1   -14.854, E3 +93365.298}
SPL {X  -160.000, Y  +585.083, Z    +0.000, E1   -14.866, E3 +93386.348}
SPL {X  -160.000, Y  +587.675, Z    +0.000, E1   -14.853, E3 +93407.139}
SPL {X  -160.000, Y  +590.216, Z    +0.000, E1   -14.864, E3 +93427.458}
SPL {X  -160.000, Y  +592.848, Z    +0.000, E1   -14.865, E3 +93448.509}
SPL {X  -160.000, Y  +595.342, Z    +0.000, E1   -14.848, E3 +93468.687}
SPL {X  -160.000, Y  +597.995, Z    +0.000, E1   -14.848, E3 +93490.027}
SPL {X  -160.000, Y  +600.731, Z    +0.000, E1   -14.846, E3 +93511.978}
SPL {X  -160.000, Y  +603.404, Z    +0.000, E1   -14.846, E3 +93533.414}
SPL {X  -160.000, Y  +605.923, Z    +0.000, E1   -14.838, E3 +93553.655}
SPL {X  -160.000, Y  +608.492, Z    +0.000, E1   -14.846, E3 +93574.259}
SPL {X  -160.000, Y  +611.345, Z    +0.000, E1   -14.856, E3 +93597.117}
SPL {X  -160.000, Y  +614.087, Z    +0.000, E1   -14.839, E3 +93619.176}
SPL {X  -160.000, Y  +616.566, Z    +0.000, E1   -14.839, E3 +93639.070}
SPL {X  -160.000, Y  +619.350, Z    +0.000, E1   -14.855, E3 +93661.358}
SPL {X  -160.000, Y  +622.198, Z    +0.000, E1   -14.846, E3 +93684.242}
SPL {X  -160.000, Y  +624.642, Z    +0.000, E1   -14.829, E3 +93703.915}
SPL {X  -160.000, Y  +627.119, Z    +0.000, E1   -14.843, E3 +93723.755}
SPL {X  -160.000, Y  +629.682, Z    +0.000, E1   -14.838, E3 +93744.324}
SPL {X  -160.000, Y  +632.223, Z    +0.000, E1   -14.841, E3 +93764.715}
SPL {X  -160.000, Y  +634.941, Z    +0.000, E1   -14.846, E3 +93786.513}
SPL {X  -160.000, Y  +637.723, Z    +0.000, E1   -14.844, E3 +93808.857}
SPL {X  -160.000, Y  +640.315, Z    +0.000, E1   -14.836, E3 +93829.654}
SPL {X  -160.000, Y  +643.085, Z    +0.000, E1   -14.865, E3 +93851.706}
SPL {X  -160.000, Y  +645.845, Z    +0.000, E1   -14.848, E3 +93873.894}
SPL {X  -160.000, Y  +648.229, Z    +0.000, E1   -14.834, E3 +93893.104}
SPL {X  -160.000, Y  +650.656, Z    +0.000, E1   -14.835, E3 +93912.660}
SPL {X  -160.000, Y  +653.134, Z    +0.000, E1   -14.827, E3 +93932.587}
SPL {X  -160.000, Y  +655.670, Z    +0.000, E1   -14.841, E3 +93952.881}
SPL {X  -160.000, Y  +658.349, Z    +0.000, E1   -14.842, E3 +93974.357}
SPL {X  -160.000, Y  +660.936, Z    +0.000, E1   -14.838, E3 +93995.109}
SPL {X  -160.000, Y  +663.567, Z    +0.000, E1   -14.845, E3 +94016.239}
SPL {X  -160.000, Y  +666.216, Z    +0.000, E1   -14.832, E3 +94037.556}
SPL {X  -159.997, Y  +668.731, Z    +0.000, E1   -14.834, E3 +94057.748}
SPL {X  -159.962, Y  +671.176, Z    +0.000, E1   -14.822, E3 +94077.459}
SPL {X  -159.895, Y  +673.507, Z    +0.000, E1   -14.821, E3 +94096.190}
SPL {X  -159.785, Y  +675.985, Z    +0.000, E1   -14.818, E3 +94116.192}
SPL {X  -159.627, Y  +678.622, Z    +0.000, E1   -14.804, E3 +94137.544}
SPL {X  -159.438, Y  +681.094, Z    +0.000, E1   -14.770, E3 +94157.716}
SPL {X  -159.262, Y  +683.054, Z    +0.000, E1   -14.719, E3 +94173.944}
ENDSPLINE

SPLINE
SPL {X  -159.661, Y  +678.114, Z    +0.000, E1    -9.575, E3 +94203.536}
SPL {X  -159.942, Y  +672.020, Z    +0.000, E1    -4.692, E3 +94222.163}
SPL {X  -160.000, Y  +664.971, Z    +0.000, E1    +0.516, E3 +94241.713}
SPL {X  -160.000, Y  +660.032, Z    +0.000, E1    +3.995, E3 +94253.656}
SPL {X  -160.000, Y  +652.280, Z    +0.000, E1    +8.913, E3 +94272.171}
SPL {X  -160.000, Y  +644.147, Z    +0.000, E1   +13.158, E3 +94295.722}
SPL {X  -160.000, Y  +641.594, Z    +0.000, E1   +13.488, E3 +94314.163}
SPL {X  -160.000, Y  +639.799, Z    +0.000, E1   +13.486, E3 +94330.073}
SPL {X  -160.000, Y  +637.896, Z    +0.000, E1   +13.493, E3 +94346.888}
SPL {X  -160.000, Y  +635.832, Z    +0.000, E1   +13.499, E3 +94365.146}
SPL {X  -160.000, Y  +633.839, Z    +0.000, E1   +13.489, E3 +94382.835}
SPL {X  -160.000, Y  +631.625, Z    +0.000, E1   +13.508, E3 +94402.376}
SPL {X  -160.000, Y  +629.417, Z    +0.000, E1   +13.491, E3 +94421.987}
SPL {X  -160.000, Y  +627.180, Z    +0.000, E1   +13.508, E3 +94441.741}
SPL {X  -160.000, Y  +624.970, Z    +0.000, E1   +13.490, E3 +94461.391}
SPL {X  -160.000, Y  +623.020, Z    +0.000, E1   +13.491, E3 +94478.621}
SPL {X  -160.000, Y  +620.888, Z    +0.000, E1   +13.501, E3 +94497.484}
SPL {X  -160.000, Y  +618.790, Z    +0.000, E1   +13.488, E3 +94516.106}
SPL {X  -160.000, Y  +616.631, Z    +0.000, E1   +13.504, E3 +94535.160}
SPL {X  -160.000, Y  +614.230, Z    +0.000, E1   +13.510, E3 +94556.356}
SPL {X  -160.000, Y  +612.132, Z    +0.000, E1   +13.485, E3 +94575.072}
SPL {X  -160.000, Y  +610.405, Z    +0.000, E1   +13.477, E3 +94590.445}
SPL {X  -160.000, Y  +608.437, Z    +0.000, E1   +13.502, E3 +94607.701}
SPL {X  -160.000, Y  +606.281, Z    +0.000, E1   +13.502, E3 +94626.718}
SPL {X  -160.000, Y  +604.124, Z    +0.000, E1   +13.513, E3 +94645.773}
SPL {X  -160.000, Y  +601.878, Z    +0.000, E1   +13.505, E3 +94665.671}
SPL {X  -160.000, Y  +599.648, Z    +0.000, E1   +13.506, E3 +94685.447}
SPL {X  -160.000, Y  +597.673, Z    +0.000, E1   +13.479, E3 +94703.121}
SPL {X  -160.000, Y  +595.601, Z    +0.000, E1   +13.499, E3 +94721.404}
SPL {X  -160.000, Y  +593.187, Z    +0.000, E1   +13.500, E3 +94742.784}
SPL {X  -160.000, Y  +591.079, Z    +0.000, E1   +13.483, E3 +94761.510}
SPL {X  -160.000, Y  +589.151, Z    +0.000, E1   +13.489, E3 +94778.561}
SPL {X  -160.000, Y  +586.908, Z    +0.000, E1   +13.501, E3 +94798.407}
SPL {X  -160.000, Y  +584.660, Z    +0.000, E1   +13.490, E3 +94818.348}
SPL {X  -160.000, Y  +582.409, Z    +0.000, E1   +13.499, E3 +94838.267}
SPL {X  -160.000, Y  +580.150, Z    +0.000, E1   +13.490, E3 +94858.313}
SPL {X  -160.000, Y  +577.953, Z    +0.000, E1   +13.493, E3 +94877.771}
SPL {X  -160.000, Y  +575.630, Z    +0.000, E1   +13.502, E3 +94898.255}
SPL {X  -160.000, Y  +573.418, Z    +0.000, E1   +13.502, E3 +94917.763}
SPL {X  -160.000, Y  +571.226, Z    +0.000, E1   +13.520, E3 +94936.972}
SPL {X  -160.000, Y  +569.166, Z    +0.000, E1   +13.512, E3 +94955.163}
SPL {X  -160.000, Y  +567.275, Z    +0.000, E1   +13.517, E3 +94971.830}
SPL {X  -160.000, Y  +565.259, Z    +0.000, E1   +13.523, E3 +94989.619}
SPL {X  -160.000, Y  +563.305, Z    +0.000, E1   +13.512, E3 +95006.957}
SPL {X  -160.000, Y  +561.240, Z    +0.000, E1   +13.521, E3 +95025.219}
SPL {X  -160.000, Y  +558.881, Z    +0.000, E1   +13.524, E3 +95046.061}
SPL {X  -160.000, Y  +556.697, Z    +0.000, E1   +13.510, E3 +95065.447}
SPL {X  -160.000, Y  +554.624, Z    +0.000, E1   +13.512, E3 +95083.778}
SPL {X  -160.000, Y  +552.465, Z    +0.000, E1   +13.514, E3 +95102.862}
SPL {X  -160.000, Y  +550.315, Z    +0.000, E1   +13.514, E3 +95121.856}
SPL {X  -160.000, Y  +548.056, Z    +0.000, E1   +13.519, E3 +95141.857}
SPL {X  -160.000, Y  +545.826, Z    +0.000, E1   +13.501, E3 +95161.735}
SPL {X  -160.000, Y  +543.677, Z    +0.000, E1   +13.502, E3 +95180.793}
SPL {X  -160.000, Y  +541.664, Z    +0.000, E1   +13.489, E3 +95198.678}
SPL {X  -160.000, Y  +539.659, Z    +0.000, E1   +13.494, E3 +95216.438}
SPL {X  -160.000, Y  +537.370, Z    +0.000, E1   +13.501, E3 +95236.677}
SPL {X  -160.000, Y  +535.056, Z    +0.000, E1   +13.506, E3 +95257.073}
SPL {X  -160.000, Y  +532.975, Z    +0.000, E1   +13.494, E3 +95275.560}
SPL {X  -160.000, Y  +530.925, Z    +0.000, E1   +13.499, E3 +95293.721}
SPL {X  -160.000, Y  +528.768, Z    +0.000, E1   +13.498, E3 +95312.823}
SPL {X  -160.000, Y  +526.547, Z    +0.000, E1   +13.499, E3 +95332.491}
SPL {X  -160.000, Y  +523.964, Z    +0.000, E1   +13.742, E3 +95351.996}
SPL {X  -160.000, Y  +513.971, Z    +0.000, E1   +18.644, E3 +95370.908}
SPL {X  -160.000, Y  +513.562, Z    +0.000, E1   +16.972, E3 +95390.784}
SPL {X  -160.000, Y  +513.358, Z    +0.000, E1   +15.267, E3 +95411.056}
SPL {X  -160.000, Y  +512.244, Z    +0.000, E1   +14.473, E3 +95429.513}
SPL {X  -160.000, Y  +509.675, Z    +0.000, E1   +14.481, E3 +95450.656}
SPL {X  -160.000, Y  +507.162, Z    +0.000, E1   +14.470, E3 +95471.396}
SPL {X  -160.000, Y  +504.735, Z    +0.000, E1   +14.473, E3 +95491.368}
SPL {X  -160.000, Y  +502.261, Z    +0.000, E1   +14.476, E3 +95511.704}
SPL {X  -160.000, Y  +499.798, Z    +0.000, E1   +14.482, E3 +95531.906}
SPL {X  -160.000, Y  +497.435, Z    +0.000, E1   +14.476, E3 +95551.383}
SPL {X  -160.000, Y  +495.089, Z    +0.000, E1   +14.475, E3 +95570.749}
SPL {X  -160.000, Y  +492.764, Z    +0.000, E1   +14.469, E3 +95589.921}
SPL {X  -160.000, Y  +490.292, Z    +0.000, E1   +14.476, E3 +95610.322}
SPL {X  -160.000, Y  +487.641, Z    +0.000, E1   +14.470, E3 +95632.218}
SPL {X  -160.000, Y  +485.054, Z    +0.000, E1   +14.460, E3 +95653.661}
SPL {X  -160.000, Y  +482.421, Z    +0.000, E1   +14.461, E3 +95675.379}
SPL {X  -160.000, Y  +480.000, Z    +0.000, E1   +14.451, E3 +95695.343}
SPL {X  -160.000, Y  +477.551, Z    +0.000, E1   +14.466, E3 +95715.472}
SPL {X  -160.000, Y  +475.253, Z    +0.000, E1   +14.450, E3 +95734.446}
SPL {X  -160.000, Y  +473.070, Z    +0.000, E1   +14.454, E3 +95752.467}
SPL {X  -160.000, Y  +470.603, Z    +0.000, E1   +14.464, E3 +95772.767}
SPL {X  -160.000, Y  +468.243, Z    +0.000, E1   +14.458, E3 +95792.166}
SPL {X  -160.000, Y  +465.791, Z    +0.000, E1   +14.475, E3 +95812.310}
SPL {X  -160.000, Y  +463.103, Z    +0.000, E1   +14.474, E3 +95834.459}
SPL {X  -160.000, Y  +460.743, Z    +0.000, E1   +14.465, E3 +95853.867}
SPL {X  -160.000, Y  +458.292, Z    +0.000, E1   +14.492, E3 +95873.867}
SPL {X  -160.000, Y  +455.874, Z    +0.000, E1   +14.484, E3 +95893.724}
SPL {X  -160.000, Y  +453.555, Z    +0.000, E1   +14.488, E3 +95912.803}
SPL {X  -160.000, Y  +451.093, Z    +0.000, E1   +14.485, E3 +95933.116}
SPL {X  -160.000, Y  +448.700, Z    +0.000, E1   +14.483, E3 +95952.805}
SPL {X  -160.000, Y  +446.277, Z    +0.000, E1   +14.485, E3 +95972.729}
SPL {X  -160.000, Y  +443.879, Z    +0.000, E1   +14.485, E3 +95992.467}
SPL {X  -160.000, Y  +441.447, Z    +0.000, E1   +14.485, E3 +96012.474}
SPL {X  -160.000, Y  +439.006, Z    +0.000, E1   +14.488, E3 +96032.557}
SPL {X  -160.000, Y  +436.311, Z    +0.000, E1   +14.498, E3 +96054.716}
SPL {X  -160.000, Y  +433.559, Z    +0.000, E1   +14.491, E3 +96077.385}
SPL {X  -160.000, Y  +431.162, Z    +0.000, E1   +14.479, E3 +96097.137}
SPL {X  -160.000, Y  +429.152, Z    +0.000, E1   +14.469, E3 +96113.718}
SPL {X  -160.000, Y  +426.863, Z    +0.000, E1   +14.490, E3 +96132.497}
SPL {X  -160.000, Y  +424.653, Z    +0.000, E1   +14.467, E3 +96150.756}
SPL {X  -160.000, Y  +422.337, Z    +0.000, E1   +14.492, E3 +96169.741}
SPL {X  -160.000, Y  +419.639, Z    +0.000, E1   +14.504, E3 +96191.780}
SPL {X  -160.000, Y  +417.127, Z    +0.000, E1   +14.501, E3 +96212.372}
SPL {X  -160.000, Y  +414.849, Z    +0.000, E1   +14.496, E3 +96231.106}
SPL {X  -160.000, Y  +412.396, Z    +0.000, E1   +14.505, E3 +96251.295}
SPL {X  -160.000, Y  +409.815, Z    +0.000, E1   +14.498, E3 +96272.549}
SPL {X  -160.000, Y  +407.614, Z    +0.000, E1   +14.484, E3 +96290.674}
SPL {X  -160.000, Y  +405.406, Z    +0.000, E1   +14.501, E3 +96308.737}
SPL {X  -160.000, Y  +402.958, Z    +0.000, E1   +14.500, E3 +96328.907}
SPL {X  -160.000, Y  +400.690, Z    +0.000, E1   +14.484, E3 +96347.619}
SPL {X  -160.000, Y  +398.391, Z    +0.000, E1   +14.502, E3 +96366.445}
SPL {X  -160.000, Y  +395.999, Z    +0.000, E1   +14.484, E3 +96386.235}
SPL {X  -160.000, Y  +393.685, Z    +0.000, E1   +14.486, E3 +96405.307}
SPL {X  -159.999, Y  +391.313, Z    +0.000, E1   +14.479, E3 +96424.889}
SPL {X  -159.970, Y  +388.900, Z    +0.000, E1   +14.480, E3 +96444.773}
SPL {X  -159.903, Y  +386.417, Z    +0.000, E1   +14.475, E3 +96465.279}
SPL {X  -159.796, Y  +383.921, Z    +0.000, E1   +14.466, E3 +96485.934}
SPL {X  -159.651, Y  +381.443, Z    +0.000, E1   +14.453, E3 +96506.482}
SPL {X  -159.474, Y  +379.042, Z    +0.000, E1   +14.434, E3 +96526.446}
SPL {X  -159.316, Y  +377.219, Z    +0.000, E1   +14.400, E3 +96541.674}
ENDSPLINE

SPLINE
SPL {X  -159.452, Y  +378.767, Z    +0.000, E1   +11.887, E3 +96562.663}
SPL {X  -159.840, Y  +384.856, Z    +0.000, E1    +7.126, E3 +96581.635}
SPL {X  -159.991, Y  +390.336, Z    +0.000, E1    +2.803, E3 +96595.458}
SPL {X  -160.000, Y  +403.532, Z    +0.000, E1    -6.523, E3 +96613.178}
SPL {X  -160.000, Y  +409.023, Z    +0.000, E1   -10.003, E3 +96623.952}
SPL {X  -160.000, Y  +418.032, Z    +0.000, E1   -14.569, E3 +96648.811}
SPL {X  -160.000, Y  +420.561, Z    +0.000, E1   -14.816, E3 +96666.291}
SPL {X  -160.000, Y  +422.801, Z    +0.000, E1   -14.823, E3 +96684.240}
SPL {X  -160.000, Y  +425.518, Z    +0.000, E1   -14.845, E3 +96706.014}
SPL {X  -160.000, Y  +428.688, Z    +0.000, E1   -14.854, E3 +96731.423}
SPL {X  -160.000, Y  +431.971, Z    +0.000, E1   -14.849, E3 +96757.891}
SPL {X  -160.000, Y  +435.345, Z    +0.000, E1   -14.857, E3 +96784.941}
SPL {X  -160.000, Y  +438.732, Z    +0.000, E1   -14.858, E3 +96812.090}
SPL {X  -160.000, Y  +441.925, Z    +0.000, E1   -14.848, E3 +96837.760}
SPL {X  -160.000, Y  +444.299, Z    +0.000, E1   -14.809, E3 +96856.945}
SPL {X  -160.000, Y  +446.229, Z    +0.000, E1   -14.820, E3 +96872.364}
SPL {X  -160.000, Y  +448.987, Z    +0.000, E1   -14.868, E3 +96894.300}
SPL {X  -160.000, Y  +452.351, Z    +0.000, E1   -14.871, E3 +96921.276}
SPL {X  -160.000, Y  +455.709, Z    +0.000, E1   -14.880, E3 +96948.091}
SPL {X  -160.000, Y  +458.189, Z    +0.000, E1   -14.832, E3 +96968.092}
SPL {X  -160.000, Y  +459.885, Z    +0.000, E1   -14.825, E3 +96981.763}
SPL {X  -160.000, Y  +462.438, Z    +0.000, E1   -14.868, E3 +97002.173}
SPL {X  -160.000, Y  +465.575, Z    +0.000, E1   -14.849, E3 +97027.481}
SPL {X  -160.000, Y  +468.581, Z    +0.000, E1   -14.841, E3 +97051.713}
SPL {X  -160.000, Y  +471.795, Z    +0.000, E1   -14.854, E3 +97077.501}
SPL {X  -160.000, Y  +475.138, Z    +0.000, E1   -14.853, E3 +97104.351}
SPL {X  -160.000, Y  +477.981, Z    +0.000, E1   -14.823, E3 +97127.272}
SPL {X  -160.000, Y  +480.658, Z    +0.000, E1   -14.835, E3 +97148.748}
SPL {X  -160.000, Y  +483.534, Z    +0.000, E1   -14.838, E3 +97171.842}
SPL {X  -160.000, Y  +486.226, Z    +0.000, E1   -14.823, E3 +97193.508}
SPL {X  -160.000, Y  +488.751, Z    +0.000, E1   -14.827, E3 +97213.780}
SPL {X  -160.000, Y  +491.612, Z    +0.000, E1   -14.844, E3 +97236.703}
SPL {X  -160.000, Y  +494.417, Z    +0.000, E1   -14.827, E3 +97259.293}
SPL {X  -160.000, Y  +496.961, Z    +0.000, E1   -14.824, E3 +97279.737}
SPL {X  -160.000, Y  +499.610, Z    +0.000, E1   -14.830, E3 +97301.010}
SPL {X  -160.000, Y  +502.268, Z    +0.000, E1   -14.832, E3 +97322.279}
SPL {X  -160.000, Y  +505.041, Z    +0.000, E1   -14.849, E3 +97344.442}
SPL {X  -160.000, Y  +507.743, Z    +0.000, E1   -14.842, E3 +97366.066}
SPL {X  -160.000, Y  +510.437, Z    +0.000, E1   -14.860, E3 +97387.579}
SPL {X  -160.000, Y  +513.179, Z    +0.000, E1   -14.849, E3 +97409.627}
SPL {X  -160.000, Y  +515.613, Z    +0.000, E1   -14.829, E3 +97429.297}
SPL {X  -160.000, Y  +518.188, Z    +0.000, E1   -14.845, E3 +97449.927}
SPL {X  -160.000, Y  +520.790, Z    +0.000, E1   -14.839, E3 +97470.755}
SPL {X  -160.000, Y  +523.469, Z    +0.000, E1   -14.855, E3 +97492.204}
SPL {X  -160.000, Y  +526.403, Z    +0.000, E1   -14.858, E3 +97515.740}
SPL {X  -160.000, Y  +529.266, Z    +0.000, E1   -14.848, E3 +97538.747}
SPL {X  -160.000, Y  +531.688, Z    +0.000, E1   -14.826, E3 +97558.297}
SPL {X  -160.000, Y  +534.214, Z    +0.000, E1   -14.841, E3 +97578.560}
SPL {X  -160.000, Y  +537.002, Z    +0.000, E1   -14.839, E3 +97600.978}
SPL {X  -160.000, Y  +539.729, Z    +0.000, E1   -14.840, E3 +97622.790}
SPL {X  -160.000, Y  +542.408, Z    +0.000, E1   -14.839, E3 +97644.343}
SPL {X  -160.000, Y  +545.014, Z    +0.000, E1   -14.831, E3 +97665.288}
SPL {X  -160.000, Y  +547.659, Z    +0.000, E1   -14.839, E3 +97686.503}
SPL {X  -160.000, Y  +550.215, Z    +0.000, E1   -14.827, E3 +97707.068}
SPL {X  -160.000, Y  +552.762, Z    +0.000, E1   -14.836, E3 +97727.486}
SPL {X  -160.000, Y  +555.331, Z    +0.000, E1   -14.837, E3 +97748.027}
SPL {X  -160.000, Y  +558.235, Z    +0.000, E1   -14.869, E3 +97771.190}
SPL {X  -160.000, Y  +561.088, Z    +0.000, E1   -14.848, E3 +97794.109}
SPL {X  -160.000, Y  +563.693, Z    +0.000, E1   -14.852, E3 +97814.969}
SPL {X  -160.000, Y  +566.560, Z    +0.000, E1   -14.865, E3 +97837.947}
SPL {X  -160.000, Y  +569.305, Z    +0.000, E1   -14.848, E3 +97859.975}
SPL {X  -160.000, Y  +571.769, Z    +0.000, E1   -14.852, E3 +97879.721}
SPL {X  -160.000, Y  +574.366, Z    +0.000, E1   -14.855, E3 +97900.508}
SPL {X  -160.000, Y  +577.037, Z    +0.000, E1   -14.859, E3 +97921.908}
SPL {X  -160.000, Y  +579.855, Z    +0.000, E1   -14.869, E3 +97944.435}
SPL {X  -160.000, Y  +582.456, Z    +0.000, E1   -14.854, E3 +97965.295}
SPL {X  -160.000, Y  +585.083, Z    +0.000, E1   -14.866, E3 +97986.345}
SPL {X  -160.000, Y  +587.675, Z    +0.000, E1   -14.853, E3 +98007.136}
SPL {X  -160.000, Y  +590.216, Z    +0.000, E1   -14.864, E3 +98027.455}
SPL {X  -160.000, Y  +592.848, Z    +0.000, E1   -14.865, E3 +98048.506}
SPL {X  -160.000, Y  +595.342, Z    +0.000, E1   -14.848, E3 +98068.684}
SPL {X  -160.000, Y  +597.995, Z    +0.000, E1   -14.848, E3 +98090.023}
SPL {X  -160.000, Y  +600.731, Z    +0.000, E1   -14.846, E3 +98111.975}
SPL {X  -160.000, Y  +603.404, Z    +0.000, E1   -14.846, E3 +98133.411}
SPL {X  -160.000, Y  +605.923, Z    +0.000, E1   -14.838, E3 +98153.652}
SPL {X  -160.000, Y  +608.492, Z    +0.000, E1   -14.846, E3 +98174.255}
SPL {X  -160.000, Y  +611.345, Z    +0.000, E1   -14.856, E3 +98197.113}
SPL {X  -160.000, Y  +614.087, Z    +0.000, E1   -14.839, E3 +98219.173}
SPL {X  -160.000, Y  +616.566, Z    +0.000, E1   -14.839, E3 +98239.067}
SPL {X  -160.000, Y  +619.350, Z    +0.000, E1   -14.855, E3 +98261.355}
SPL {X  -160.000, Y  +622.198, Z    +0.000, E1   -14.846, E3 +98284.239}
SPL {X  -160.000, Y  +624.642, Z    +0.000, E1   -14.829, E3 +98303.912}
SPL {X  -160.000, Y  +627.119, Z    +0.000, E1   -14.843, E3 +98323.752}
SPL {X  -160.000, Y  +629.682, Z    +0.000, E1   -14.838, E3 +98344.321}
SPL {X  -160.000, Y  +632.223, Z    +0.000, E1   -14.841, E3 +98364.712}
SPL {X  -160.000, Y  +634.941, Z    +0.000, E1   -14.846, E3 +98386.509}
SPL {X  -160.000, Y  +637.723, Z    +0.000, E1   -14.844, E3 +98408.854}
SPL {X  -160.000, Y  +640.315, Z    +0.000, E1   -14.836, E3 +98429.651}
SPL {X  -160.000, Y  +643.085, Z    +0.000, E1   -14.865, E3 +98451.703}
SPL {X  -160.000, Y  +645.845, Z    +0.000, E1   -14.848, E3 +98473.891}
SPL {X  -160.000, Y  +648.229, Z    +0.000, E1   -14.834, E3 +98493.101}
SPL {X  -160.000, Y  +650.656, Z    +0.000, E1   -14.835, E3 +98512.657}
SPL {X  -160.000, Y  +653.134, Z    +0.000, E1   -14.827, E3 +98532.584}
SPL {X  -160.000, Y  +655.670, Z    +0.000, E1   -14.841, E3 +98552.878}
SPL {X  -160.000, Y  +658.349, Z    +0.000, E1   -14.842, E3 +98574.354}
SPL {X  -160.000, Y  +660.936, Z    +0.000, E1   -14.838, E3 +98595.106}
SPL {X  -160.000, Y  +663.567, Z    +0.000, E1   -14.845, E3 +98616.236}
SPL {X  -160.000, Y  +666.216, Z    +0.000, E1   -14.832, E3 +98637.552}
SPL {X  -159.997, Y  +668.731, Z    +0.000, E1   -14.834, E3 +98657.744}
SPL {X  -159.962, Y  +671.176, Z    +0.000, E1   -14.822, E3 +98677.456}
SPL {X  -159.895, Y  +673.507, Z    +0.000, E1   -14.821, E3 +98696.187}
SPL {X  -159.785, Y  +675.985, Z    +0.000, E1   -14.818, E3 +98716.188}
SPL {X  -159.627, Y  +678.622, Z    +0.000, E1   -14.804, E3 +98737.541}
SPL {X  -159.438, Y  +681.094, Z    +0.000, E1   -14.770, E3 +98757.713}
SPL {X  -159.262, Y  +683.054, Z    +0.000, E1   -14.719, E3 +98773.941}
ENDSPLINE

SPLINE
SPL {X  -159.661, Y  +678.114, Z    +0.000, E1    -9.575, E3 +98803.533}
SPL {X  -159.942, Y  +672.020, Z    +0.000, E1    -4.692, E3 +98822.160}
SPL {X  -160.000, Y  +664.971, Z    +0.000, E1    +0.516, E3 +98841.710}
SPL {X  -160.000, Y  +660.032, Z    +0.000, E1    +3.995, E3 +98853.653}
SPL {X  -160.000, Y  +652.280, Z    +0.000, E1    +8.913, E3 +98872.168}
SPL {X  -160.000, Y  +644.147, Z    +0.000, E1   +13.158, E3 +98895.718}
SPL {X  -160.000, Y  +641.594, Z    +0.000, E1   +13.488, E3 +98914.159}
SPL {X  -160.000, Y  +639.799, Z    +0.000, E1   +13.486, E3 +98930.069}
SPL {X  -160.000, Y  +637.896, Z    +0.000, E1   +13.493, E3 +98946.884}
SPL {X  -160.000, Y  +635.832, Z    +0.000, E1   +13.499, E3 +98965.143}
SPL {X  -160.000, Y  +633.839, Z    +0.000, E1   +13.489, E3 +98982.832}
SPL {X  -160.000, Y  +631.625, Z    +0.000, E1   +13.508, E3 +99002.373}
SPL {X  -160.000, Y  +629.417, Z    +0.000, E1   +13.491, E3 +99021.984}
SPL {X  -160.000, Y  +627.180, Z    +0.000, E1   +13.508, E3 +99041.738}
SPL {X  -160.000, Y  +624.970, Z    +0.000, E1   +13.490, E3 +99061.388}
SPL {X  -160.000, Y  +623.020, Z    +0.000, E1   +13.491, E3 +99078.618}
SPL {X  -160.000, Y  +620.888, Z    +0.000, E1   +13.501, E3 +99097.480}
SPL {X  -160.000, Y  +618.790, Z    +0.000, E1   +13.488, E3 +99116.103}
SPL {X  -160.000, Y  +616.631, Z    +0.000, E1   +13.504, E3 +99135.156}
SPL {X  -160.000, Y  +614.230, Z    +0.000, E1   +13.510, E3 +99156.352}
SPL {X  -160.000, Y  +612.132, Z    +0.000, E1   +13.485, E3 +99175.069}
SPL {X  -160.000, Y  +610.405, Z    +0.000, E1   +13.477, E3 +99190.442}
SPL {X  -160.000, Y  +608.437, Z    +0.000, E1   +13.502, E3 +99207.697}
SPL {X  -160.000, Y  +606.281, Z    +0.000, E1   +13.502, E3 +99226.715}
SPL {X  -160.000, Y  +604.124, Z    +0.000, E1   +13.513, E3 +99245.770}
SPL {X  -160.000, Y  +601.878, Z    +0.000, E1   +13.505, E3 +99265.667}
SPL {X  -160.000, Y  +599.648, Z    +0.000, E1   +13.506, E3 +99285.444}
SPL {X  -160.000, Y  +597.673, Z    +0.000, E1   +13.479, E3 +99303.118}
SPL {X  -160.000, Y  +595.601, Z    +0.000, E1   +13.499, E3 +99321.401}
SPL {X  -160.000, Y  +593.187, Z    +0.000, E1   +13.500, E3 +99342.781}
SPL {X  -160.000, Y  +591.079, Z    +0.000, E1   +13.483, E3 +99361.507}
SPL {X  -160.000, Y  +589.151, Z    +0.000, E1   +13.489, E3 +99378.558}
SPL {X  -160.000, Y  +586.908, Z    +0.000, E1   +13.501, E3 +99398.404}
SPL {X  -160.000, Y  +584.660, Z    +0.000, E1   +13.490, E3 +99418.345}
SPL {X  -160.000, Y  +582.409, Z    +0.000, E1   +13.499, E3 +99438.263}
SPL {X  -160.000, Y  +580.150, Z    +0.000, E1   +13.490, E3 +99458.310}
SPL {X  -160.000, Y  +577.953, Z    +0.000, E1   +13.493, E3 +99477.768}
SPL {X  -160.000, Y  +575.630, Z    +0.000, E1   +13.502, E3 +99498.252}
SPL {X  -160.000, Y  +573.418, Z    +0.000, E1   +13.502, E3 +99517.760}
SPL {X  -160.000, Y  +571.226, Z    +0.000, E1   +13.520, E3 +99536.969}
SPL {X  -160.000, Y  +569.166, Z    +0.000, E1   +13.512, E3 +99555.159}
SPL {X  -160.000, Y  +567.275, Z    +0.000, E1   +13.517, E3 +99571.827}
SPL {X  -160.000, Y  +565.259, Z    +0.000, E1   +13.523, E3 +99589.616}
SPL {X  -160.000, Y  +563.305, Z    +0.000, E1   +13.512, E3 +99606.954}
SPL {X  -160.000, Y  +561.240, Z    +0.000, E1   +13.521, E3 +99625.216}
SPL {X  -160.000, Y  +558.881, Z    +0.000, E1   +13.524, E3 +99646.058}
SPL {X  -160.000, Y  +556.697, Z    +0.000, E1   +13.510, E3 +99665.444}
SPL {X  -160.000, Y  +554.624, Z    +0.000, E1   +13.512, E3 +99683.775}
SPL {X  -160.000, Y  +552.465, Z    +0.000, E1   +13.514, E3 +99702.859}
SPL {X  -160.000, Y  +550.315, Z    +0.000, E1   +13.514, E3 +99721.853}
SPL {X  -160.000, Y  +548.056, Z    +0.000, E1   +13.519, E3 +99741.854}
SPL {X  -160.000, Y  +545.826, Z    +0.000, E1   +13.501, E3 +99761.732}
SPL {X  -160.000, Y  +543.677, Z    +0.000, E1   +13.502, E3 +99780.790}
SPL {X  -160.000, Y  +541.664, Z    +0.000, E1   +13.489, E3 +99798.675}
SPL {X  -160.000, Y  +539.659, Z    +0.000, E1   +13.494, E3 +99816.435}
SPL {X  -160.000, Y  +537.370, Z    +0.000, E1   +13.501, E3 +99836.674}
SPL {X  -160.000, Y  +535.056, Z    +0.000, E1   +13.506, E3 +99857.070}
SPL {X  -160.000, Y  +532.975, Z    +0.000, E1   +13.494, E3 +99875.556}
SPL {X  -160.000, Y  +530.925, Z    +0.000, E1   +13.499, E3 +99893.718}
SPL {X  -160.000, Y  +528.768, Z    +0.000, E1   +13.498, E3 +99912.819}
SPL {X  -160.000, Y  +526.547, Z    +0.000, E1   +13.499, E3 +99932.488}
SPL {X  -160.000, Y  +523.964, Z    +0.000, E1   +13.742, E3 +99951.993}
SPL {X  -160.000, Y  +513.971, Z    +0.000, E1   +18.644, E3 +99970.905}
SPL {X  -160.000, Y  +513.562, Z    +0.000, E1   +16.972, E3 +99990.781}
SPL {X  -160.000, Y  +513.358, Z    +0.000, E1   +15.267, E3 +100011.053}
SPL {X  -160.000, Y  +512.244, Z    +0.000, E1   +14.473, E3 +100029.510}
SPL {X  -160.000, Y  +509.675, Z    +0.000, E1   +14.481, E3 +100050.653}
SPL {X  -160.000, Y  +507.162, Z    +0.000, E1   +14.470, E3 +100071.393}
SPL {X  -160.000, Y  +504.735, Z    +0.000, E1   +14.473, E3 +100091.364}
SPL {X  -160.000, Y  +502.261, Z    +0.000, E1   +14.476, E3 +100111.701}
SPL {X  -160.000, Y  +499.798, Z    +0.000, E1   +14.482, E3 +100131.903}
SPL {X  -160.000, Y  +497.435, Z    +0.000, E1   +14.476, E3 +100151.379}
SPL {X  -160.000, Y  +495.089, Z    +0.000, E1   +14.475, E3 +100170.746}
SPL {X  -160.000, Y  +492.764, Z    +0.000, E1   +14.469, E3 +100189.918}
SPL {X  -160.000, Y  +490.292, Z    +0.000, E1   +14.476, E3 +100210.319}
SPL {X  -160.000, Y  +487.641, Z    +0.000, E1   +14.470, E3 +100232.215}
SPL {X  -160.000, Y  +485.054, Z    +0.000, E1   +14.460, E3 +100253.657}
SPL {X  -160.000, Y  +482.421, Z    +0.000, E1   +14.461, E3 +100275.376}
SPL {X  -160.000, Y  +480.000, Z    +0.000, E1   +14.451, E3 +100295.340}
SPL {X  -160.000, Y  +477.551, Z    +0.000, E1   +14.466, E3 +100315.468}
SPL {X  -160.000, Y  +475.253, Z    +0.000, E1   +14.450, E3 +100334.443}
SPL {X  -160.000, Y  +473.070, Z    +0.000, E1   +14.454, E3 +100352.464}
SPL {X  -160.000, Y  +470.603, Z    +0.000, E1   +14.464, E3 +100372.764}
SPL {X  -160.000, Y  +468.243, Z    +0.000, E1   +14.458, E3 +100392.163}
SPL {X  -160.000, Y  +465.791, Z    +0.000, E1   +14.475, E3 +100412.307}
SPL {X  -160.000, Y  +463.103, Z    +0.000, E1   +14.474, E3 +100434.456}
SPL {X  -160.000, Y  +460.743, Z    +0.000, E1   +14.465, E3 +100453.864}
SPL {X  -160.000, Y  +458.292, Z    +0.000, E1   +14.492, E3 +100473.863}
SPL {X  -160.000, Y  +455.874, Z    +0.000, E1   +14.484, E3 +100493.721}
SPL {X  -160.000, Y  +453.555, Z    +0.000, E1   +14.488, E3 +100512.800}
SPL {X  -160.000, Y  +451.093, Z    +0.000, E1   +14.485, E3 +100533.112}
SPL {X  -160.000, Y  +448.700, Z    +0.000, E1   +14.483, E3 +100552.802}
SPL {X  -160.000, Y  +446.277, Z    +0.000, E1   +14.485, E3 +100572.725}
SPL {X  -160.000, Y  +443.879, Z    +0.000, E1   +14.485, E3 +100592.464}
SPL {X  -160.000, Y  +441.447, Z    +0.000, E1   +14.485, E3 +100612.471}
SPL {X  -160.000, Y  +439.006, Z    +0.000, E1   +14.488, E3 +100632.554}
SPL {X  -160.000, Y  +436.311, Z    +0.000, E1   +14.498, E3 +100654.713}
SPL {X  -160.000, Y  +433.559, Z    +0.000, E1   +14.491, E3 +100677.382}
SPL {X  -160.000, Y  +431.162, Z    +0.000, E1   +14.479, E3 +100697.134}
SPL {X  -160.000, Y  +429.152, Z    +0.000, E1   +14.469, E3 +100713.715}
SPL {X  -160.000, Y  +426.863, Z    +0.000, E1   +14.490, E3 +100732.494}
SPL {X  -160.000, Y  +424.653, Z    +0.000, E1   +14.467, E3 +100750.753}
SPL {X  -160.000, Y  +422.337, Z    +0.000, E1   +14.492, E3 +100769.737}
SPL {X  -160.000, Y  +419.639, Z    +0.000, E1   +14.504, E3 +100791.777}
SPL {X  -160.000, Y  +417.127, Z    +0.000, E1   +14.501, E3 +100812.369}
SPL {X  -160.000, Y  +414.849, Z    +0.000, E1   +14.496, E3 +100831.103}
SPL {X  -160.000, Y  +412.396, Z    +0.000, E1   +14.505, E3 +100851.292}
SPL {X  -160.000, Y  +409.815, Z    +0.000, E1   +14.498, E3 +100872.546}
SPL {X  -160.000, Y  +407.614, Z    +0.000, E1   +14.484, E3 +100890.671}
SPL {X  -160.000, Y  +405.406, Z    +0.000, E1   +14.501, E3 +100908.734}
SPL {X  -160.000, Y  +402.958, Z    +0.000, E1   +14.500, E3 +100928.904}
SPL {X  -160.000, Y  +400.690, Z    +0.000, E1   +14.484, E3 +100947.616}
SPL {X  -160.000, Y  +398.391, Z    +0.000, E1   +14.502, E3 +100966.442}
SPL {X  -160.000, Y  +395.999, Z    +0.000, E1   +14.484, E3 +100986.232}
SPL {X  -160.000, Y  +393.685, Z    +0.000, E1   +14.486, E3 +101005.304}
SPL {X  -159.999, Y  +391.313, Z    +0.000, E1   +14.479, E3 +101024.886}
SPL {X  -159.970, Y  +388.900, Z    +0.000, E1   +14.480, E3 +101044.770}
SPL {X  -159.903, Y  +386.417, Z    +0.000, E1   +14.475, E3 +101065.275}
SPL {X  -159.796, Y  +383.921, Z    +0.000, E1   +14.466, E3 +101085.931}
SPL {X  -159.651, Y  +381.443, Z    +0.000, E1   +14.453, E3 +101106.479}
SPL {X  -159.474, Y  +379.042, Z    +0.000, E1   +14.434, E3 +101126.443}
SPL {X  -159.316, Y  +377.219, Z    +0.000, E1   +14.400, E3 +101141.671}
ENDSPLINE

SPLINE
SPL {X  -159.452, Y  +378.767, Z    +0.000, E1   +11.887, E3 +101162.660}
SPL {X  -159.840, Y  +384.856, Z    +0.000, E1    +7.126, E3 +101181.632}
SPL {X  -159.991, Y  +390.336, Z    +0.000, E1    +2.803, E3 +101195.455}
SPL {X  -160.000, Y  +403.532, Z    +0.000, E1    -6.523, E3 +101213.175}
SPL {X  -160.000, Y  +409.023, Z    +0.000, E1   -10.003, E3 +101223.949}
SPL {X  -160.000, Y  +418.032, Z    +0.000, E1   -14.569, E3 +101248.808}
SPL {X  -160.000, Y  +420.561, Z    +0.000, E1   -14.816, E3 +101266.288}
SPL {X  -160.000, Y  +422.801, Z    +0.000, E1   -14.823, E3 +101284.237}
SPL {X  -160.000, Y  +425.518, Z    +0.000, E1   -14.845, E3 +101306.011}
SPL {X  -160.000, Y  +428.688, Z    +0.000, E1   -14.854, E3 +101331.419}
SPL {X  -160.000, Y  +431.971, Z    +0.000, E1   -14.849, E3 +101357.888}
SPL {X  -160.000, Y  +435.345, Z    +0.000, E1   -14.857, E3 +101384.938}
SPL {X  -160.000, Y  +438.732, Z    +0.000, E1   -14.858, E3 +101412.087}
SPL {X  -160.000, Y  +441.925, Z    +0.000, E1   -14.848, E3 +101437.757}
SPL {X  -160.000, Y  +444.299, Z    +0.000, E1   -14.809, E3 +101456.942}
SPL {X  -160.000, Y  +446.229, Z    +0.000, E1   -14.820, E3 +101472.361}
SPL {X  -160.000, Y  +448.987, Z    +0.000, E1   -14.868, E3 +101494.297}
SPL {X  -160.000, Y  +452.351, Z    +0.000, E1   -14.871, E3 +101521.273}
SPL {X  -160.000, Y  +455.709, Z    +0.000, E1   -14.880, E3 +101548.087}
SPL {X  -160.000, Y  +458.189, Z    +0.000, E1   -14.832, E3 +101568.089}
SPL {X  -160.000, Y  +459.885, Z    +0.000, E1   -14.825, E3 +101581.760}
SPL {X  -160.000, Y  +462.438, Z    +0.000, E1   -14.868, E3 +101602.170}
SPL {X  -160.000, Y  +465.575, Z    +0.000, E1   -14.849, E3 +101627.478}
SPL {X  -160.000, Y  +468.581, Z    +0.000, E1   -14.841, E3 +101651.710}
SPL {X  -160.000, Y  +471.795, Z    +0.000, E1   -14.854, E3 +101677.498}
SPL {X  -160.000, Y  +475.138, Z    +0.000, E1   -14.853, E3 +101704.348}
SPL {X  -160.000, Y  +477.981, Z    +0.000, E1   -14.823, E3 +101727.268}
SPL {X  -160.000, Y  +480.658, Z    +0.000, E1   -14.835, E3 +101748.744}
SPL {X  -160.000, Y  +483.534, Z    +0.000, E1   -14.838, E3 +101771.839}
SPL {X  -160.000, Y  +486.226, Z    +0.000, E1   -14.823, E3 +101793.504}
SPL {X  -160.000, Y  +488.751, Z    +0.000, E1   -14.827, E3 +101813.777}
SPL {X  -160.000, Y  +491.612, Z    +0.000, E1   -14.844, E3 +101836.699}
SPL {X  -160.000, Y  +494.417, Z    +0.000, E1   -14.827, E3 +101859.290}
SPL {X  -160.000, Y  +496.961, Z    +0.000, E1   -14.824, E3 +101879.734}
SPL {X  -160.000, Y  +499.610, Z    +0.000, E1   -14.830, E3 +101901.007}
SPL {X  -160.000, Y  +502.268, Z    +0.000, E1   -14.832, E3 +101922.276}
SPL {X  -160.000, Y  +505.041, Z    +0.000, E1   -14.849, E3 +101944.439}
SPL {X  -160.000, Y  +507.743, Z    +0.000, E1   -14.842, E3 +101966.062}
SPL {X  -160.000, Y  +510.437, Z    +0.000, E1   -14.860, E3 +101987.576}
SPL {X  -160.000, Y  +513.179, Z    +0.000, E1   -14.849, E3 +102009.624}
SPL {X  -160.000, Y  +515.613, Z    +0.000, E1   -14.829, E3 +102029.294}
SPL {X  -160.000, Y  +518.188, Z    +0.000, E1   -14.845, E3 +102049.923}
SPL {X  -160.000, Y  +520.790, Z    +0.000, E1   -14.839, E3 +102070.752}
SPL {X  -160.000, Y  +523.469, Z    +0.000, E1   -14.855, E3 +102092.200}
SPL {X  -160.000, Y  +526.403, Z    +0.000, E1   -14.858, E3 +102115.737}
SPL {X  -160.000, Y  +529.266, Z    +0.000, E1   -14.848, E3 +102138.744}
SPL {X  -160.000, Y  +531.688, Z    +0.000, E1   -14.826, E3 +102158.294}
SPL {X  -160.000, Y  +534.214, Z    +0.000, E1   -14.841, E3 +102178.557}
SPL {X  -160.000, Y  +537.002, Z    +0.000, E1   -14.839, E3 +102200.975}
SPL {X  -160.000, Y  +539.729, Z    +0.000, E1   -14.840, E3 +102222.787}
SPL {X  -160.000, Y  +542.408, Z    +0.000, E1   -14.839, E3 +102244.340}
SPL {X  -160.000, Y  +545.014, Z    +0.000, E1   -14.831, E3 +102265.285}
SPL {X  -160.000, Y  +547.659, Z    +0.000, E1   -14.839, E3 +102286.499}
SPL {X  -160.000, Y  +550.215, Z    +0.000, E1   -14.827, E3 +102307.064}
SPL {X  -160.000, Y  +552.762, Z    +0.000, E1   -14.836, E3 +102327.483}
SPL {X  -160.000, Y  +555.331, Z    +0.000, E1   -14.837, E3 +102348.024}
SPL {X  -160.000, Y  +558.235, Z    +0.000, E1   -14.869, E3 +102371.187}
SPL {X  -160.000, Y  +561.088, Z    +0.000, E1   -14.848, E3 +102394.106}
SPL {X  -160.000, Y  +563.693, Z    +0.000, E1   -14.852, E3 +102414.966}
SPL {X  -160.000, Y  +566.560, Z    +0.000, E1   -14.865, E3 +102437.944}
SPL {X  -160.000, Y  +569.305, Z    +0.000, E1   -14.848, E3 +102459.972}
SPL {X  -160.000, Y  +571.769, Z    +0.000, E1   -14.852, E3 +102479.718}
SPL {X  -160.000, Y  +574.366, Z    +0.000, E1   -14.855, E3 +102500.505}
SPL {X  -160.000, Y  +577.037, Z    +0.000, E1   -14.859, E3 +102521.905}
SPL {X  -160.000, Y  +579.855, Z    +0.000, E1   -14.869, E3 +102544.432}
SPL {X  -160.000, Y  +582.456, Z    +0.000, E1   -14.854, E3 +102565.292}
SPL {X  -160.000, Y  +585.083, Z    +0.000, E1   -14.866, E3 +102586.341}
SPL {X  -160.000, Y  +587.675, Z    +0.000, E1   -14.853, E3 +102607.132}
SPL {X  -160.000, Y  +590.216, Z    +0.000, E1   -14.864, E3 +102627.452}
SPL {X  -160.000, Y  +592.848, Z    +0.000, E1   -14.865, E3 +102648.503}
SPL {X  -160.000, Y  +595.342, Z    +0.000, E1   -14.848, E3 +102668.680}
SPL {X  -160.000, Y  +597.995, Z    +0.000, E1   -14.848, E3 +102690.020}
SPL {X  -160.000, Y  +600.731, Z    +0.000, E1   -14.846, E3 +102711.972}
SPL {X  -160.000, Y  +603.404, Z    +0.000, E1   -14.846, E3 +102733.408}
SPL {X  -160.000, Y  +605.923, Z    +0.000, E1   -14.838, E3 +102753.648}
SPL {X  -160.000, Y  +608.492, Z    +0.000, E1   -14.846, E3 +102774.252}
SPL {X  -160.000, Y  +611.345, Z    +0.000, E1   -14.856, E3 +102797.110}
SPL {X  -160.000, Y  +614.087, Z    +0.000, E1   -14.839, E3 +102819.170}
SPL {X  -160.000, Y  +616.566, Z    +0.000, E1   -14.839, E3 +102839.063}
SPL {X  -160.000, Y  +619.350, Z    +0.000, E1   -14.855, E3 +102861.351}
SPL {X  -160.000, Y  +622.198, Z    +0.000, E1   -14.846, E3 +102884.236}
SPL {X  -160.000, Y  +624.642, Z    +0.000, E1   -14.829, E3 +102903.909}
SPL {X  -160.000, Y  +627.119, Z    +0.000, E1   -14.843, E3 +102923.748}
SPL {X  -160.000, Y  +629.682, Z    +0.000, E1   -14.838, E3 +102944.317}
SPL {X  -160.000, Y  +632.223, Z    +0.000, E1   -14.841, E3 +102964.709}
SPL {X  -160.000, Y  +634.941, Z    +0.000, E1   -14.846, E3 +102986.506}
SPL {X  -160.000, Y  +637.723, Z    +0.000, E1   -14.844, E3 +103008.851}
SPL {X  -160.000, Y  +640.315, Z    +0.000, E1   -14.836, E3 +103029.648}
SPL {X  -160.000, Y  +643.085, Z    +0.000, E1   -14.865, E3 +103051.700}
SPL {X  -160.000, Y  +645.845, Z    +0.000, E1   -14.848, E3 +103073.888}
SPL {X  -160.000, Y  +648.229, Z    +0.000, E1   -14.834, E3 +103093.097}
SPL {X  -160.000, Y  +650.656, Z    +0.000, E1   -14.835, E3 +103112.654}
SPL {X  -160.000, Y  +653.134, Z    +0.000, E1   -14.827, E3 +103132.581}
SPL {X  -160.000, Y  +655.670, Z    +0.000, E1   -14.841, E3 +103152.875}
SPL {X  -160.000, Y  +658.349, Z    +0.000, E1   -14.842, E3 +103174.351}
SPL {X  -160.000, Y  +660.936, Z    +0.000, E1   -14.838, E3 +103195.102}
SPL {X  -160.000, Y  +663.567, Z    +0.000, E1   -14.845, E3 +103216.233}
SPL {X  -160.000, Y  +666.216, Z    +0.000, E1   -14.832, E3 +103237.549}
SPL {X  -159.997, Y  +668.731, Z    +0.000, E1   -14.834, E3 +103257.741}
SPL {X  -159.962, Y  +671.176, Z    +0.000, E1   -14.822, E3 +103277.452}
SPL {X  -159.895, Y  +673.507, Z    +0.000, E1   -14.821, E3 +103296.184}
SPL {X  -159.785, Y  +675.985, Z    +0.000, E1   -14.818, E3 +103316.185}
SPL {X  -159.627, Y  +678.622, Z    +0.000, E1   -14.804, E3 +103337.538}
SPL {X  -159.438, Y  +681.094, Z    +0.000, E1   -14.770, E3 +103357.710}
SPL {X  -159.262, Y  +683.054, Z    +0.000, E1   -14.719, E3 +103373.938}
ENDSPLINE

SPLINE
SPL {X  -159.661, Y  +678.114, Z    +0.000, E1    -9.575, E3 +103403.530}
SPL {X  -159.942, Y  +672.020, Z    +0.000, E1    -4.692, E3 +103422.157}
SPL {X  -160.000, Y  +664.971, Z    +0.000, E1    +0.516, E3 +103441.707}
SPL {X  -160.000, Y  +660.032, Z    +0.000, E1    +3.995, E3 +103453.650}
SPL {X  -160.000, Y  +652.280, Z    +0.000, E1    +8.913, E3 +103472.165}
SPL {X  -160.000, Y  +644.147, Z    +0.000, E1   +13.158, E3 +103495.715}
SPL {X  -160.000, Y  +641.594, Z    +0.000, E1   +13.488, E3 +103514.156}
SPL {X  -160.000, Y  +639.799, Z    +0.000, E1   +13.486, E3 +103530.066}
SPL {X  -160.000, Y  +637.896, Z    +0.000, E1   +13.493, E3 +103546.881}
SPL {X  -160.000, Y  +635.832, Z    +0.000, E1   +13.499, E3 +103565.140}
SPL {X  -160.000, Y  +633.839, Z    +0.000, E1   +13.489, E3 +103582.829}
SPL {X  -160.000, Y  +631.625, Z    +0.000, E1   +13.508, E3 +103602.370}
SPL {X  -160.000, Y  +629.417, Z    +0.000, E1   +13.491, E3 +103621.981}
SPL {X  -160.000, Y  +627.180, Z    +0.000, E1   +13.508, E3 +103641.735}
SPL {X  -160.000, Y  +624.970, Z    +0.000, E1   +13.490, E3 +103661.385}
SPL {X  -160.000, Y  +623.020, Z    +0.000, E1   +13.491, E3 +103678.615}
SPL {X  -160.000, Y  +620.888, Z    +0.000, E1   +13.501, E3 +103697.477}
SPL {X  -160.000, Y  +618.790, Z    +0.000, E1   +13.488, E3 +103716.100}
SPL {X  -160.000, Y  +616.631, Z    +0.000, E1   +13.504, E3 +103735.153}
SPL {X  -160.000, Y  +614.230, Z    +0.000, E1   +13.510, E3 +103756.349}
SPL {X  -160.000, Y  +612.132, Z    +0.000, E1   +13.485, E3 +103775.065}
SPL {X  -160.000, Y  +610.405, Z    +0.000, E1   +13.477, E3 +103790.439}
SPL {X  -160.000, Y  +608.437, Z    +0.000, E1   +13.502, E3 +103807.694}
SPL {X  -160.000, Y  +606.281, Z    +0.000, E1   +13.502, E3 +103826.712}
SPL {X  -160.000, Y  +604.124, Z    +0.000, E1   +13.513, E3 +103845.767}
SPL {X  -160.000, Y  +601.878, Z    +0.000, E1   +13.505, E3 +103865.664}
SPL {X  -160.000, Y  +599.648, Z    +0.000, E1   +13.506, E3 +103885.441}
SPL {X  -160.000, Y  +597.673, Z    +0.000, E1   +13.479, E3 +103903.115}
SPL {X  -160.000, Y  +595.601, Z    +0.000, E1   +13.499, E3 +103921.398}
SPL {X  -160.000, Y  +593.187, Z    +0.000, E1   +13.500, E3 +103942.778}
SPL {X  -160.000, Y  +591.079, Z    +0.000, E1   +13.483, E3 +103961.504}
SPL {X  -160.000, Y  +589.151, Z    +0.000, E1   +13.489, E3 +103978.555}
SPL {X  -160.000, Y  +586.908, Z    +0.000, E1   +13.501, E3 +103998.400}
SPL {X  -160.000, Y  +584.660, Z    +0.000, E1   +13.490, E3 +104018.342}
SPL {X  -160.000, Y  +582.409, Z    +0.000, E1   +13.499, E3 +104038.260}
SPL {X  -160.000, Y  +580.150, Z    +0.000, E1   +13.490, E3 +104058.307}
SPL {X  -160.000, Y  +577.953, Z    +0.000, E1   +13.493, E3 +104077.765}
SPL {X  -160.000, Y  +575.630, Z    +0.000, E1   +13.502, E3 +104098.249}
SPL {X  -160.000, Y  +573.418, Z    +0.000, E1   +13.502, E3 +104117.757}
SPL {X  -160.000, Y  +571.226, Z    +0.000, E1   +13.520, E3 +104136.966}
SPL {X  -160.000, Y  +569.166, Z    +0.000, E1   +13.512, E3 +104155.156}
SPL {X  -160.000, Y  +567.275, Z    +0.000, E1   +13.517, E3 +104171.824}
SPL {X  -160.000, Y  +565.259, Z    +0.000, E1   +13.523, E3 +104189.613}
SPL {X  -160.000, Y  +563.305, Z    +0.000, E1   +13.512, E3 +104206.951}
SPL {X  -160.000, Y  +561.240, Z    +0.000, E1   +13.521, E3 +104225.213}
SPL {X  -160.000, Y  +558.881, Z    +0.000, E1   +13.524, E3 +104246.055}
SPL {X  -160.000, Y  +556.697, Z    +0.000, E1   +13.510, E3 +104265.441}
SPL {X  -160.000, Y  +554.624, Z    +0.000, E1   +13.512, E3 +104283.772}
SPL {X  -160.000, Y  +552.465, Z    +0.000, E1   +13.514, E3 +104302.856}
SPL {X  -160.000, Y  +550.315, Z    +0.000, E1   +13.514, E3 +104321.850}
SPL {X  -160.000, Y  +548.056, Z    +0.000, E1   +13.519, E3 +104341.851}
SPL {X  -160.000, Y  +545.826, Z    +0.000, E1   +13.501, E3 +104361.728}
SPL {X  -160.000, Y  +543.677, Z    +0.000, E1   +13.502, E3 +104380.786}
SPL {X  -160.000, Y  +541.664, Z    +0.000, E1   +13.489, E3 +104398.672}
SPL {X  -160.000, Y  +539.659, Z    +0.000, E1   +13.494, E3 +104416.432}
SPL {X  -160.000, Y  +537.370, Z    +0.000, E1   +13.501, E3 +104436.671}
SPL {X  -160.000, Y  +535.056, Z    +0.000, E1   +13.506, E3 +104457.066}
SPL {X  -160.000, Y  +532.975, Z    +0.000, E1   +13.494, E3 +104475.553}
SPL {X  -160.000, Y  +530.925, Z    +0.000, E1   +13.499, E3 +104493.715}
SPL {X  -160.000, Y  +528.768, Z    +0.000, E1   +13.498, E3 +104512.816}
SPL {X  -160.000, Y  +526.547, Z    +0.000, E1   +13.499, E3 +104532.485}
SPL {X  -160.000, Y  +523.964, Z    +0.000, E1   +13.742, E3 +104551.989}
SPL {X  -160.000, Y  +513.971, Z    +0.000, E1   +18.644, E3 +104570.901}
SPL {X  -160.000, Y  +513.562, Z    +0.000, E1   +16.972, E3 +104590.778}
SPL {X  -160.000, Y  +513.358, Z    +0.000, E1   +15.267, E3 +104611.050}
SPL {X  -160.000, Y  +512.244, Z    +0.000, E1   +14.473, E3 +104629.506}
SPL {X  -160.000, Y  +509.675, Z    +0.000, E1   +14.481, E3 +104650.650}
SPL {X  -160.000, Y  +507.162, Z    +0.000, E1   +14.470, E3 +104671.390}
SPL {X  -160.000, Y  +504.735, Z    +0.000, E1   +14.473, E3 +104691.361}
SPL {X  -160.000, Y  +502.261, Z    +0.000, E1   +14.476, E3 +104711.697}
SPL {X  -160.000, Y  +499.798, Z    +0.000, E1   +14.482, E3 +104731.900}
SPL {X  -160.000, Y  +497.435, Z    +0.000, E1   +14.476, E3 +104751.376}
SPL {X  -160.000, Y  +495.089, Z    +0.000, E1   +14.475, E3 +104770.743}
SPL {X  -160.000, Y  +492.764, Z    +0.000, E1   +14.469, E3 +104789.915}
SPL {X  -160.000, Y  +490.292, Z    +0.000, E1   +14.476, E3 +104810.316}
SPL {X  -160.000, Y  +487.641, Z    +0.000, E1   +14.470, E3 +104832.212}
SPL {X  -160.000, Y  +485.054, Z    +0.000, E1   +14.460, E3 +104853.654}
SPL {X  -160.000, Y  +482.421, Z    +0.000, E1   +14.461, E3 +104875.373}
SPL {X  -160.000, Y  +480.000, Z    +0.000, E1   +14.451, E3 +104895.337}
SPL {X  -160.000, Y  +477.551, Z    +0.000, E1   +14.466, E3 +104915.465}
SPL {X  -160.000, Y  +475.253, Z    +0.000, E1   +14.450, E3 +104934.439}
SPL {X  -160.000, Y  +473.070, Z    +0.000, E1   +14.454, E3 +104952.460}
SPL {X  -160.000, Y  +470.603, Z    +0.000, E1   +14.464, E3 +104972.760}
SPL {X  -160.000, Y  +468.243, Z    +0.000, E1   +14.458, E3 +104992.160}
SPL {X  -160.000, Y  +465.791, Z    +0.000, E1   +14.475, E3 +105012.304}
SPL {X  -160.000, Y  +463.103, Z    +0.000, E1   +14.474, E3 +105034.453}
SPL {X  -160.000, Y  +460.743, Z    +0.000, E1   +14.465, E3 +105053.861}
SPL {X  -160.000, Y  +458.292, Z    +0.000, E1   +14.492, E3 +105073.860}
SPL {X  -160.000, Y  +455.874, Z    +0.000, E1   +14.484, E3 +105093.718}
SPL {X  -160.000, Y  +453.555, Z    +0.000, E1   +14.488, E3 +105112.797}
SPL {X  -160.000, Y  +451.093, Z    +0.000, E1   +14.485, E3 +105133.109}
SPL {X  -160.000, Y  +448.700, Z    +0.000, E1   +14.483, E3 +105152.799}
SPL {X  -160.000, Y  +446.277, Z    +0.000, E1   +14.485, E3 +105172.722}
SPL {X  -160.000, Y  +443.879, Z    +0.000, E1   +14.485, E3 +105192.460}
SPL {X  -160.000, Y  +441.447, Z    +0.000, E1   +14.485, E3 +105212.468}
SPL {X  -160.000, Y  +439.006, Z    +0.000, E1   +14.488, E3 +105232.551}
SPL {X  -160.000, Y  +436.311, Z    +0.000, E1   +14.498, E3 +105254.710}
SPL {X  -160.000, Y  +433.559, Z    +0.000, E1   +14.491, E3 +105277.379}
SPL {X  -160.000, Y  +431.162, Z    +0.000, E1   +14.479, E3 +105297.130}
SPL {X  -160.000, Y  +429.152, Z    +0.000, E1   +14.469, E3 +105313.712}
SPL {X  -160.000, Y  +426.863, Z    +0.000, E1   +14.490, E3 +105332.491}
SPL {X  -160.000, Y  +424.653, Z    +0.000, E1   +14.467, E3 +105350.750}
SPL {X  -160.000, Y  +422.337, Z    +0.000, E1   +14.492, E3 +105369.734}
SPL {X  -160.000, Y  +419.639, Z    +0.000, E1   +14.504, E3 +105391.774}
SPL {X  -160.000, Y  +417.127, Z    +0.000, E1   +14.501, E3 +105412.365}
SPL {X  -160.000, Y  +414.849, Z    +0.000, E1   +14.496, E3 +105431.099}
SPL {X  -160.000, Y  +412.396, Z    +0.000, E1   +14.505, E3 +105451.288}
SPL {X  -160.000, Y  +409.815, Z    +0.000, E1   +14.498, E3 +105472.543}
SPL {X  -160.000, Y  +407.614, Z    +0.000, E1   +14.484, E3 +105490.668}
SPL {X  -160.000, Y  +405.406, Z    +0.000, E1   +14.501, E3 +105508.731}
SPL {X  -160.000, Y  +402.958, Z    +0.000, E1   +14.500, E3 +105528.901}
SPL {X  -160.000, Y  +400.690, Z    +0.000, E1   +14.484, E3 +105547.613}
SPL {X  -160.000, Y  +398.391, Z    +0.000, E1   +14.502, E3 +105566.439}
SPL {X  -160.000, Y  +395.999, Z    +0.000, E1   +14.484, E3 +105586.228}
SPL {X  -160.000, Y  +393.685, Z    +0.000, E1   +14.486, E3 +105605.301}
SPL {X  -159.999, Y  +391.313, Z    +0.000, E1   +14.479, E3 +105624.883}
SPL {X  -159.970, Y  +388.900, Z    +0.000, E1   +14.480, E3 +105644.767}
SPL {X  -159.903, Y  +386.417, Z    +0.000, E1   +14.475, E3 +105665.272}
SPL {X  -159.796, Y  +383.921, Z    +0.000, E1   +14.466, E3 +105685.928}
SPL {X  -159.651, Y  +381.443, Z    +0.000, E1   +14.453, E3 +105706.475}
SPL {X  -159.474, Y  +379.042, Z    +0.000, E1   +14.434, E3 +105726.439}
SPL {X  -159.316, Y  +377.219, Z    +0.000, E1   +14.400, E3 +105741.668}
ENDSPLINE

